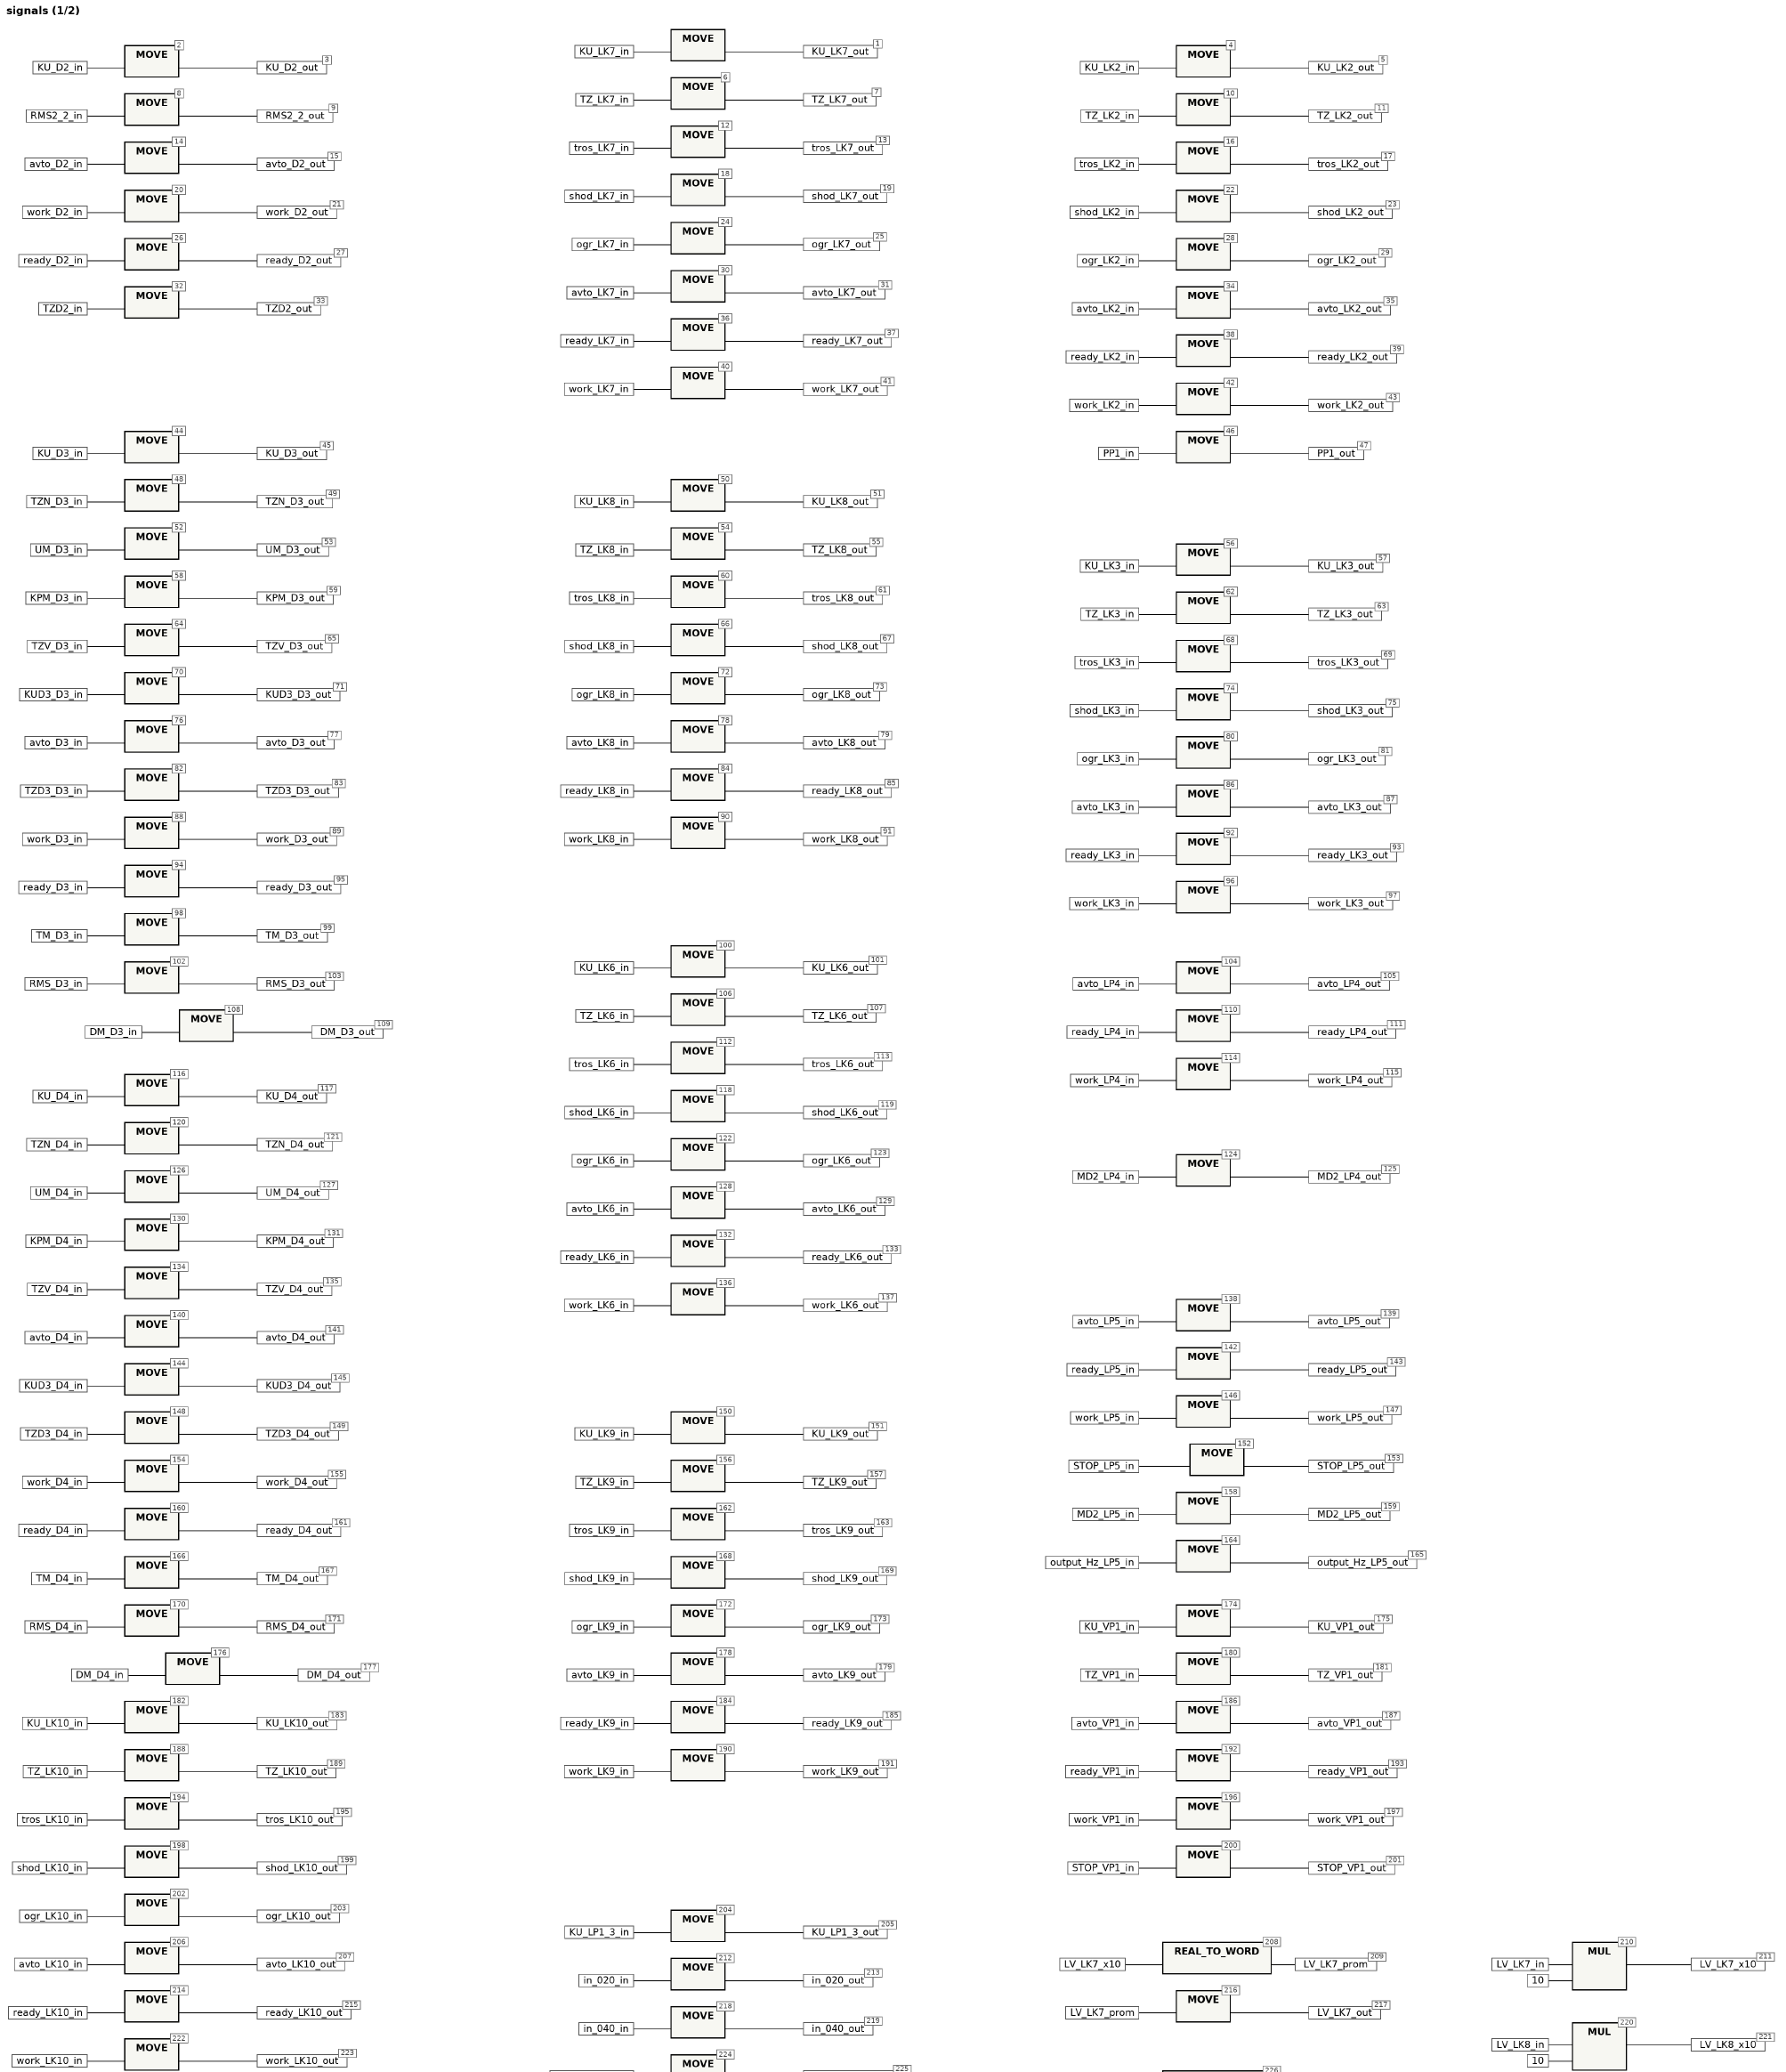
[picture p55: signals (CFC)]
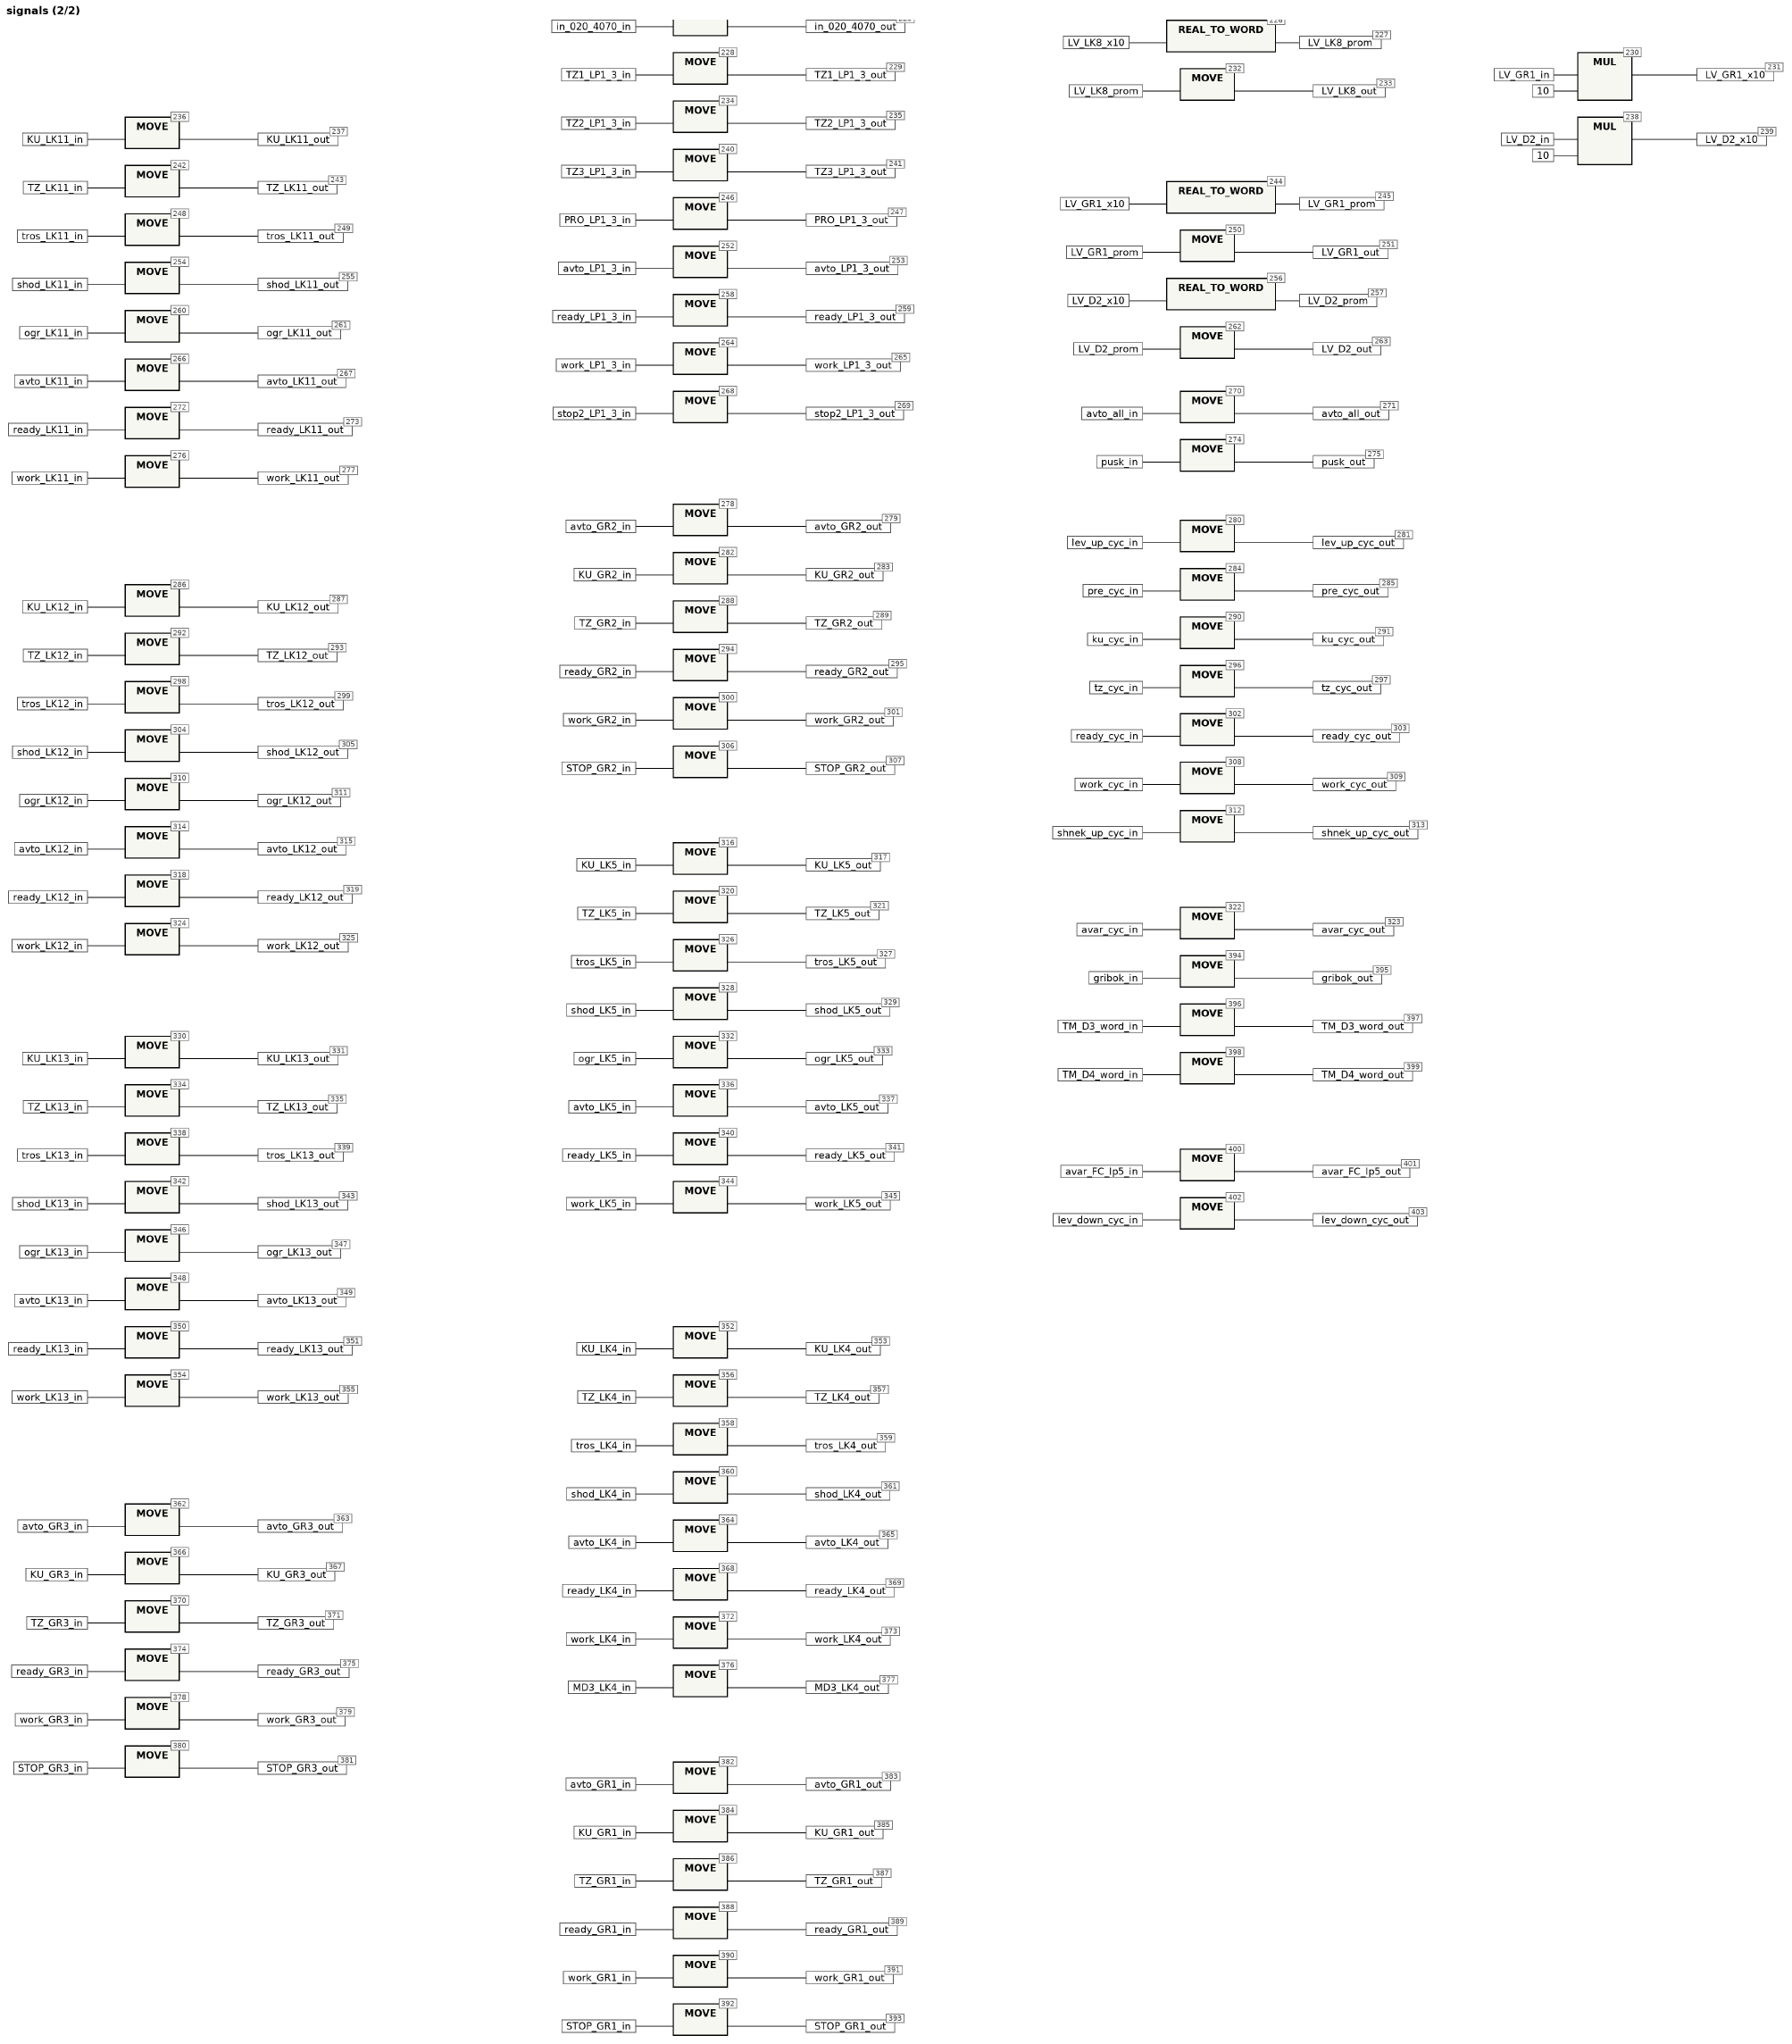
_CFC_ (* Continuous Function Chart, elements in execution order *)
#0 MOVE(KU_LK7_in)
#1 KU_LK7_out <= #0
#2 MOVE(KU_D2_in)
#3 KU_D2_out <= #2
#4 MOVE(KU_LK2_in)
#5 KU_LK2_out <= #4
#6 MOVE(TZ_LK7_in)
#7 TZ_LK7_out <= #6
#8 MOVE(RMS2_2_in)
#9 RMS2_2_out <= #8
#10 MOVE(TZ_LK2_in)
#11 TZ_LK2_out <= #10
#12 MOVE(tros_LK7_in)
#13 tros_LK7_out <= #12
#14 MOVE(avto_D2_in)
#15 avto_D2_out <= #14
#16 MOVE(tros_LK2_in)
#17 tros_LK2_out <= #16
#18 MOVE(shod_LK7_in)
#19 shod_LK7_out <= #18
#20 MOVE(work_D2_in)
#21 work_D2_out <= #20
#22 MOVE(shod_LK2_in)
#23 shod_LK2_out <= #22
#24 MOVE(ogr_LK7_in)
#25 ogr_LK7_out <= #24
#26 MOVE(ready_D2_in)
#27 ready_D2_out <= #26
#28 MOVE(ogr_LK2_in)
#29 ogr_LK2_out <= #28
#30 MOVE(avto_LK7_in)
#31 avto_LK7_out <= #30
#32 MOVE(TZD2_in)
#33 TZD2_out <= #32
#34 MOVE(avto_LK2_in)
#35 avto_LK2_out <= #34
#36 MOVE(ready_LK7_in)
#37 ready_LK7_out <= #36
#38 MOVE(ready_LK2_in)
#39 ready_LK2_out <= #38
#40 MOVE(work_LK7_in)
#41 work_LK7_out <= #40
#42 MOVE(work_LK2_in)
#43 work_LK2_out <= #42
#44 MOVE(KU_D3_in)
#45 KU_D3_out <= #44
#46 MOVE(PP1_in)
#47 PP1_out <= #46
#48 MOVE(TZN_D3_in)
#49 TZN_D3_out <= #48
#50 MOVE(KU_LK8_in)
#51 KU_LK8_out <= #50
#52 MOVE(UM_D3_in)
#53 UM_D3_out <= #52
#54 MOVE(TZ_LK8_in)
#55 TZ_LK8_out <= #54
#56 MOVE(KU_LK3_in)
#57 KU_LK3_out <= #56
#58 MOVE(KPM_D3_in)
#59 KPM_D3_out <= #58
#60 MOVE(tros_LK8_in)
#61 tros_LK8_out <= #60
#62 MOVE(TZ_LK3_in)
#63 TZ_LK3_out <= #62
#64 MOVE(TZV_D3_in)
#65 TZV_D3_out <= #64
#66 MOVE(shod_LK8_in)
#67 shod_LK8_out <= #66
#68 MOVE(tros_LK3_in)
#69 tros_LK3_out <= #68
#70 MOVE(KUD3_D3_in)
#71 KUD3_D3_out <= #70
#72 MOVE(ogr_LK8_in)
#73 ogr_LK8_out <= #72
#74 MOVE(shod_LK3_in)
#75 shod_LK3_out <= #74
#76 MOVE(avto_D3_in)
#77 avto_D3_out <= #76
#78 MOVE(avto_LK8_in)
#79 avto_LK8_out <= #78
#80 MOVE(ogr_LK3_in)
#81 ogr_LK3_out <= #80
#82 MOVE(TZD3_D3_in)
#83 TZD3_D3_out <= #82
#84 MOVE(ready_LK8_in)
#85 ready_LK8_out <= #84
#86 MOVE(avto_LK3_in)
#87 avto_LK3_out <= #86
#88 MOVE(work_D3_in)
#89 work_D3_out <= #88
#90 MOVE(work_LK8_in)
#91 work_LK8_out <= #90
#92 MOVE(ready_LK3_in)
#93 ready_LK3_out <= #92
#94 MOVE(ready_D3_in)
#95 ready_D3_out <= #94
#96 MOVE(work_LK3_in)
#97 work_LK3_out <= #96
#98 MOVE(TM_D3_in)
#99 TM_D3_out <= #98
#100 MOVE(KU_LK6_in)
#101 KU_LK6_out <= #100
#102 MOVE(RMS_D3_in)
#103 RMS_D3_out <= #102
#104 MOVE(avto_LP4_in)
#105 avto_LP4_out <= #104
#106 MOVE(TZ_LK6_in)
#107 TZ_LK6_out <= #106
#108 MOVE(DM_D3_in)
#109 DM_D3_out <= #108
#110 MOVE(ready_LP4_in)
#111 ready_LP4_out <= #110
#112 MOVE(tros_LK6_in)
#113 tros_LK6_out <= #112
#114 MOVE(work_LP4_in)
#115 work_LP4_out <= #114
#116 MOVE(KU_D4_in)
#117 KU_D4_out <= #116
#118 MOVE(shod_LK6_in)
#119 shod_LK6_out <= #118
#120 MOVE(TZN_D4_in)
#121 TZN_D4_out <= #120
#122 MOVE(ogr_LK6_in)
#123 ogr_LK6_out <= #122
#124 MOVE(MD2_LP4_in)
#125 MD2_LP4_out <= #124
#126 MOVE(UM_D4_in)
#127 UM_D4_out <= #126
#128 MOVE(avto_LK6_in)
#129 avto_LK6_out <= #128
#130 MOVE(KPM_D4_in)
#131 KPM_D4_out <= #130
#132 MOVE(ready_LK6_in)
#133 ready_LK6_out <= #132
#134 MOVE(TZV_D4_in)
#135 TZV_D4_out <= #134
#136 MOVE(work_LK6_in)
#137 work_LK6_out <= #136
#138 MOVE(avto_LP5_in)
#139 avto_LP5_out <= #138
#140 MOVE(avto_D4_in)
#141 avto_D4_out <= #140
#142 MOVE(ready_LP5_in)
#143 ready_LP5_out <= #142
#144 MOVE(KUD3_D4_in)
#145 KUD3_D4_out <= #144
#146 MOVE(work_LP5_in)
#147 work_LP5_out <= #146
#148 MOVE(TZD3_D4_in)
#149 TZD3_D4_out <= #148
#150 MOVE(KU_LK9_in)
#151 KU_LK9_out <= #150
#152 MOVE(STOP_LP5_in)
#153 STOP_LP5_out <= #152
#154 MOVE(work_D4_in)
#155 work_D4_out <= #154
#156 MOVE(TZ_LK9_in)
#157 TZ_LK9_out <= #156
#158 MOVE(MD2_LP5_in)
#159 MD2_LP5_out <= #158
#160 MOVE(ready_D4_in)
#161 ready_D4_out <= #160
#162 MOVE(tros_LK9_in)
#163 tros_LK9_out <= #162
#164 MOVE(output_Hz_LP5_in)
#165 output_Hz_LP5_out <= #164
#166 MOVE(TM_D4_in)
#167 TM_D4_out <= #166
#168 MOVE(shod_LK9_in)
#169 shod_LK9_out <= #168
#170 MOVE(RMS_D4_in)
#171 RMS_D4_out <= #170
#172 MOVE(ogr_LK9_in)
#173 ogr_LK9_out <= #172
#174 MOVE(KU_VP1_in)
#175 KU_VP1_out <= #174
#176 MOVE(DM_D4_in)
#177 DM_D4_out <= #176
#178 MOVE(avto_LK9_in)
#179 avto_LK9_out <= #178
#180 MOVE(TZ_VP1_in)
#181 TZ_VP1_out <= #180
#182 MOVE(KU_LK10_in)
#183 KU_LK10_out <= #182
#184 MOVE(ready_LK9_in)
#185 ready_LK9_out <= #184
#186 MOVE(avto_VP1_in)
#187 avto_VP1_out <= #186
#188 MOVE(TZ_LK10_in)
#189 TZ_LK10_out <= #188
#190 MOVE(work_LK9_in)
#191 work_LK9_out <= #190
#192 MOVE(ready_VP1_in)
#193 ready_VP1_out <= #192
#194 MOVE(tros_LK10_in)
#195 tros_LK10_out <= #194
#196 MOVE(work_VP1_in)
#197 work_VP1_out <= #196
#198 MOVE(shod_LK10_in)
#199 shod_LK10_out <= #198
#200 MOVE(STOP_VP1_in)
#201 STOP_VP1_out <= #200
#202 MOVE(ogr_LK10_in)
#203 ogr_LK10_out <= #202
#204 MOVE(KU_LP1_3_in)
#205 KU_LP1_3_out <= #204
#206 MOVE(avto_LK10_in)
#207 avto_LK10_out <= #206
#208 REAL_TO_WORD(LV_LK7_x10)
#209 LV_LK7_prom <= #208
#210 MUL(LV_LK7_in, 10)
#211 LV_LK7_x10 <= #210
#212 MOVE(in_020_in)
#213 in_020_out <= #212
#214 MOVE(ready_LK10_in)
#215 ready_LK10_out <= #214
#216 MOVE(LV_LK7_prom)
#217 LV_LK7_out <= #216
#218 MOVE(in_040_in)
#219 in_040_out <= #218
#220 MUL(LV_LK8_in, 10)
#221 LV_LK8_x10 <= #220
#222 MOVE(work_LK10_in)
#223 work_LK10_out <= #222
#224 MOVE(in_020_4070_in)
#225 in_020_4070_out <= #224
#226 REAL_TO_WORD(LV_LK8_x10)
#227 LV_LK8_prom <= #226
#228 MOVE(TZ1_LP1_3_in)
#229 TZ1_LP1_3_out <= #228
#230 MUL(LV_GR1_in, 10)
#231 LV_GR1_x10 <= #230
#232 MOVE(LV_LK8_prom)
#233 LV_LK8_out <= #232
#234 MOVE(TZ2_LP1_3_in)
#235 TZ2_LP1_3_out <= #234
#236 MOVE(KU_LK11_in)
#237 KU_LK11_out <= #236
#238 MUL(LV_D2_in, 10)
#239 LV_D2_x10 <= #238
#240 MOVE(TZ3_LP1_3_in)
#241 TZ3_LP1_3_out <= #240
#242 MOVE(TZ_LK11_in)
#243 TZ_LK11_out <= #242
#244 REAL_TO_WORD(LV_GR1_x10)
#245 LV_GR1_prom <= #244
#246 MOVE(PRO_LP1_3_in)
#247 PRO_LP1_3_out <= #246
#248 MOVE(tros_LK11_in)
#249 tros_LK11_out <= #248
#250 MOVE(LV_GR1_prom)
#251 LV_GR1_out <= #250
#252 MOVE(avto_LP1_3_in)
#253 avto_LP1_3_out <= #252
#254 MOVE(shod_LK11_in)
#255 shod_LK11_out <= #254
#256 REAL_TO_WORD(LV_D2_x10)
#257 LV_D2_prom <= #256
#258 MOVE(ready_LP1_3_in)
#259 ready_LP1_3_out <= #258
#260 MOVE(ogr_LK11_in)
#261 ogr_LK11_out <= #260
#262 MOVE(LV_D2_prom)
#263 LV_D2_out <= #262
#264 MOVE(work_LP1_3_in)
#265 work_LP1_3_out <= #264
#266 MOVE(avto_LK11_in)
#267 avto_LK11_out <= #266
#268 MOVE(stop2_LP1_3_in)
#269 stop2_LP1_3_out <= #268
#270 MOVE(avto_all_in)
#271 avto_all_out <= #270
#272 MOVE(ready_LK11_in)
#273 ready_LK11_out <= #272
#274 MOVE(pusk_in)
#275 pusk_out <= #274
#276 MOVE(work_LK11_in)
#277 work_LK11_out <= #276
#278 MOVE(avto_GR2_in)
#279 avto_GR2_out <= #278
#280 MOVE(lev_up_cyc_in)
#281 lev_up_cyc_out <= #280
#282 MOVE(KU_GR2_in)
#283 KU_GR2_out <= #282
#284 MOVE(pre_cyc_in)
#285 pre_cyc_out <= #284
#286 MOVE(KU_LK12_in)
#287 KU_LK12_out <= #286
#288 MOVE(TZ_GR2_in)
#289 TZ_GR2_out <= #288
#290 MOVE(ku_cyc_in)
#291 ku_cyc_out <= #290
#292 MOVE(TZ_LK12_in)
#293 TZ_LK12_out <= #292
#294 MOVE(ready_GR2_in)
#295 ready_GR2_out <= #294
#296 MOVE(tz_cyc_in)
#297 tz_cyc_out <= #296
#298 MOVE(tros_LK12_in)
#299 tros_LK12_out <= #298
#300 MOVE(work_GR2_in)
#301 work_GR2_out <= #300
#302 MOVE(ready_cyc_in)
#303 ready_cyc_out <= #302
#304 MOVE(shod_LK12_in)
#305 shod_LK12_out <= #304
#306 MOVE(STOP_GR2_in)
#307 STOP_GR2_out <= #306
#308 MOVE(work_cyc_in)
#309 work_cyc_out <= #308
#310 MOVE(ogr_LK12_in)
#311 ogr_LK12_out <= #310
#312 MOVE(shnek_up_cyc_in)
#313 shnek_up_cyc_out <= #312
#314 MOVE(avto_LK12_in)
#315 avto_LK12_out <= #314
#316 MOVE(KU_LK5_in)
#317 KU_LK5_out <= #316
#318 MOVE(ready_LK12_in)
#319 ready_LK12_out <= #318
#320 MOVE(TZ_LK5_in)
#321 TZ_LK5_out <= #320
#322 MOVE(avar_cyc_in)
#323 avar_cyc_out <= #322
#324 MOVE(work_LK12_in)
#325 work_LK12_out <= #324
#326 MOVE(tros_LK5_in)
#327 tros_LK5_out <= #326
#328 MOVE(shod_LK5_in)
#329 shod_LK5_out <= #328
#330 MOVE(KU_LK13_in)
#331 KU_LK13_out <= #330
#332 MOVE(ogr_LK5_in)
#333 ogr_LK5_out <= #332
#334 MOVE(TZ_LK13_in)
#335 TZ_LK13_out <= #334
#336 MOVE(avto_LK5_in)
#337 avto_LK5_out <= #336
#338 MOVE(tros_LK13_in)
#339 tros_LK13_out <= #338
#340 MOVE(ready_LK5_in)
#341 ready_LK5_out <= #340
#342 MOVE(shod_LK13_in)
#343 shod_LK13_out <= #342
#344 MOVE(work_LK5_in)
#345 work_LK5_out <= #344
#346 MOVE(ogr_LK13_in)
#347 ogr_LK13_out <= #346
#348 MOVE(avto_LK13_in)
#349 avto_LK13_out <= #348
#350 MOVE(ready_LK13_in)
#351 ready_LK13_out <= #350
#352 MOVE(KU_LK4_in)
#353 KU_LK4_out <= #352
#354 MOVE(work_LK13_in)
#355 work_LK13_out <= #354
#356 MOVE(TZ_LK4_in)
#357 TZ_LK4_out <= #356
#358 MOVE(tros_LK4_in)
#359 tros_LK4_out <= #358
#360 MOVE(shod_LK4_in)
#361 shod_LK4_out <= #360
#362 MOVE(avto_GR3_in)
#363 avto_GR3_out <= #362
#364 MOVE(avto_LK4_in)
#365 avto_LK4_out <= #364
#366 MOVE(KU_GR3_in)
#367 KU_GR3_out <= #366
#368 MOVE(ready_LK4_in)
#369 ready_LK4_out <= #368
#370 MOVE(TZ_GR3_in)
#371 TZ_GR3_out <= #370
#372 MOVE(work_LK4_in)
#373 work_LK4_out <= #372
#374 MOVE(ready_GR3_in)
#375 ready_GR3_out <= #374
#376 MOVE(MD3_LK4_in)
#377 MD3_LK4_out <= #376
#378 MOVE(work_GR3_in)
#379 work_GR3_out <= #378
#380 MOVE(STOP_GR3_in)
#381 STOP_GR3_out <= #380
#382 MOVE(avto_GR1_in)
#383 avto_GR1_out <= #382
#384 MOVE(KU_GR1_in)
#385 KU_GR1_out <= #384
#386 MOVE(TZ_GR1_in)
#387 TZ_GR1_out <= #386
#388 MOVE(ready_GR1_in)
#389 ready_GR1_out <= #388
#390 MOVE(work_GR1_in)
#391 work_GR1_out <= #390
#392 MOVE(STOP_GR1_in)
#393 STOP_GR1_out <= #392
#394 MOVE(gribok_in)
#395 gribok_out <= #394
#396 MOVE(TM_D3_word_in)
#397 TM_D3_word_out <= #396
#398 MOVE(TM_D4_word_in)
#399 TM_D4_word_out <= #398
#400 MOVE(avar_FC_lp5_in)
#401 avar_FC_lp5_out <= #400
#402 MOVE(lev_down_cyc_in)
#403 lev_down_cyc_out <= #402
_END_CFC_
(* the same logic as Structured Text *)
KU_LK7_out := KU_LK7_in;
KU_D2_out := KU_D2_in;
KU_LK2_out := KU_LK2_in;
TZ_LK7_out := TZ_LK7_in;
RMS2_2_out := RMS2_2_in;
TZ_LK2_out := TZ_LK2_in;
tros_LK7_out := tros_LK7_in;
avto_D2_out := avto_D2_in;
tros_LK2_out := tros_LK2_in;
shod_LK7_out := shod_LK7_in;
work_D2_out := work_D2_in;
shod_LK2_out := shod_LK2_in;
ogr_LK7_out := ogr_LK7_in;
ready_D2_out := ready_D2_in;
ogr_LK2_out := ogr_LK2_in;
avto_LK7_out := avto_LK7_in;
TZD2_out := TZD2_in;
avto_LK2_out := avto_LK2_in;
ready_LK7_out := ready_LK7_in;
ready_LK2_out := ready_LK2_in;
work_LK7_out := work_LK7_in;
work_LK2_out := work_LK2_in;
KU_D3_out := KU_D3_in;
PP1_out := PP1_in;
TZN_D3_out := TZN_D3_in;
KU_LK8_out := KU_LK8_in;
UM_D3_out := UM_D3_in;
TZ_LK8_out := TZ_LK8_in;
KU_LK3_out := KU_LK3_in;
KPM_D3_out := KPM_D3_in;
tros_LK8_out := tros_LK8_in;
TZ_LK3_out := TZ_LK3_in;
TZV_D3_out := TZV_D3_in;
shod_LK8_out := shod_LK8_in;
tros_LK3_out := tros_LK3_in;
KUD3_D3_out := KUD3_D3_in;
ogr_LK8_out := ogr_LK8_in;
shod_LK3_out := shod_LK3_in;
avto_D3_out := avto_D3_in;
avto_LK8_out := avto_LK8_in;
ogr_LK3_out := ogr_LK3_in;
TZD3_D3_out := TZD3_D3_in;
ready_LK8_out := ready_LK8_in;
avto_LK3_out := avto_LK3_in;
work_D3_out := work_D3_in;
work_LK8_out := work_LK8_in;
ready_LK3_out := ready_LK3_in;
ready_D3_out := ready_D3_in;
work_LK3_out := work_LK3_in;
TM_D3_out := TM_D3_in;
KU_LK6_out := KU_LK6_in;
RMS_D3_out := RMS_D3_in;
avto_LP4_out := avto_LP4_in;
TZ_LK6_out := TZ_LK6_in;
DM_D3_out := DM_D3_in;
ready_LP4_out := ready_LP4_in;
tros_LK6_out := tros_LK6_in;
work_LP4_out := work_LP4_in;
KU_D4_out := KU_D4_in;
shod_LK6_out := shod_LK6_in;
TZN_D4_out := TZN_D4_in;
ogr_LK6_out := ogr_LK6_in;
MD2_LP4_out := MD2_LP4_in;
UM_D4_out := UM_D4_in;
avto_LK6_out := avto_LK6_in;
KPM_D4_out := KPM_D4_in;
ready_LK6_out := ready_LK6_in;
TZV_D4_out := TZV_D4_in;
work_LK6_out := work_LK6_in;
avto_LP5_out := avto_LP5_in;
avto_D4_out := avto_D4_in;
ready_LP5_out := ready_LP5_in;
KUD3_D4_out := KUD3_D4_in;
work_LP5_out := work_LP5_in;
TZD3_D4_out := TZD3_D4_in;
KU_LK9_out := KU_LK9_in;
STOP_LP5_out := STOP_LP5_in;
work_D4_out := work_D4_in;
TZ_LK9_out := TZ_LK9_in;
MD2_LP5_out := MD2_LP5_in;
ready_D4_out := ready_D4_in;
tros_LK9_out := tros_LK9_in;
output_Hz_LP5_out := output_Hz_LP5_in;
TM_D4_out := TM_D4_in;
shod_LK9_out := shod_LK9_in;
RMS_D4_out := RMS_D4_in;
ogr_LK9_out := ogr_LK9_in;
KU_VP1_out := KU_VP1_in;
DM_D4_out := DM_D4_in;
avto_LK9_out := avto_LK9_in;
TZ_VP1_out := TZ_VP1_in;
KU_LK10_out := KU_LK10_in;
ready_LK9_out := ready_LK9_in;
avto_VP1_out := avto_VP1_in;
TZ_LK10_out := TZ_LK10_in;
work_LK9_out := work_LK9_in;
ready_VP1_out := ready_VP1_in;
tros_LK10_out := tros_LK10_in;
work_VP1_out := work_VP1_in;
shod_LK10_out := shod_LK10_in;
STOP_VP1_out := STOP_VP1_in;
ogr_LK10_out := ogr_LK10_in;
KU_LP1_3_out := KU_LP1_3_in;
avto_LK10_out := avto_LK10_in;
LV_LK7_prom := REAL_TO_WORD(LV_LK7_x10);
LV_LK7_x10 := LV_LK7_in * 10;
in_020_out := in_020_in;
ready_LK10_out := ready_LK10_in;
LV_LK7_out := LV_LK7_prom;
in_040_out := in_040_in;
LV_LK8_x10 := LV_LK8_in * 10;
work_LK10_out := work_LK10_in;
in_020_4070_out := in_020_4070_in;
LV_LK8_prom := REAL_TO_WORD(LV_LK8_x10);
TZ1_LP1_3_out := TZ1_LP1_3_in;
LV_GR1_x10 := LV_GR1_in * 10;
LV_LK8_out := LV_LK8_prom;
TZ2_LP1_3_out := TZ2_LP1_3_in;
KU_LK11_out := KU_LK11_in;
LV_D2_x10 := LV_D2_in * 10;
TZ3_LP1_3_out := TZ3_LP1_3_in;
TZ_LK11_out := TZ_LK11_in;
LV_GR1_prom := REAL_TO_WORD(LV_GR1_x10);
PRO_LP1_3_out := PRO_LP1_3_in;
tros_LK11_out := tros_LK11_in;
LV_GR1_out := LV_GR1_prom;
avto_LP1_3_out := avto_LP1_3_in;
shod_LK11_out := shod_LK11_in;
LV_D2_prom := REAL_TO_WORD(LV_D2_x10);
ready_LP1_3_out := ready_LP1_3_in;
ogr_LK11_out := ogr_LK11_in;
LV_D2_out := LV_D2_prom;
work_LP1_3_out := work_LP1_3_in;
avto_LK11_out := avto_LK11_in;
stop2_LP1_3_out := stop2_LP1_3_in;
avto_all_out := avto_all_in;
ready_LK11_out := ready_LK11_in;
pusk_out := pusk_in;
work_LK11_out := work_LK11_in;
avto_GR2_out := avto_GR2_in;
lev_up_cyc_out := lev_up_cyc_in;
KU_GR2_out := KU_GR2_in;
pre_cyc_out := pre_cyc_in;
KU_LK12_out := KU_LK12_in;
TZ_GR2_out := TZ_GR2_in;
ku_cyc_out := ku_cyc_in;
TZ_LK12_out := TZ_LK12_in;
ready_GR2_out := ready_GR2_in;
tz_cyc_out := tz_cyc_in;
tros_LK12_out := tros_LK12_in;
work_GR2_out := work_GR2_in;
ready_cyc_out := ready_cyc_in;
shod_LK12_out := shod_LK12_in;
STOP_GR2_out := STOP_GR2_in;
work_cyc_out := work_cyc_in;
ogr_LK12_out := ogr_LK12_in;
shnek_up_cyc_out := shnek_up_cyc_in;
avto_LK12_out := avto_LK12_in;
KU_LK5_out := KU_LK5_in;
ready_LK12_out := ready_LK12_in;
TZ_LK5_out := TZ_LK5_in;
avar_cyc_out := avar_cyc_in;
work_LK12_out := work_LK12_in;
tros_LK5_out := tros_LK5_in;
shod_LK5_out := shod_LK5_in;
KU_LK13_out := KU_LK13_in;
ogr_LK5_out := ogr_LK5_in;
TZ_LK13_out := TZ_LK13_in;
avto_LK5_out := avto_LK5_in;
tros_LK13_out := tros_LK13_in;
ready_LK5_out := ready_LK5_in;
shod_LK13_out := shod_LK13_in;
work_LK5_out := work_LK5_in;
ogr_LK13_out := ogr_LK13_in;
avto_LK13_out := avto_LK13_in;
ready_LK13_out := ready_LK13_in;
KU_LK4_out := KU_LK4_in;
work_LK13_out := work_LK13_in;
TZ_LK4_out := TZ_LK4_in;
tros_LK4_out := tros_LK4_in;
shod_LK4_out := shod_LK4_in;
avto_GR3_out := avto_GR3_in;
avto_LK4_out := avto_LK4_in;
KU_GR3_out := KU_GR3_in;
ready_LK4_out := ready_LK4_in;
TZ_GR3_out := TZ_GR3_in;
work_LK4_out := work_LK4_in;
ready_GR3_out := ready_GR3_in;
MD3_LK4_out := MD3_LK4_in;
work_GR3_out := work_GR3_in;
STOP_GR3_out := STOP_GR3_in;
avto_GR1_out := avto_GR1_in;
KU_GR1_out := KU_GR1_in;
TZ_GR1_out := TZ_GR1_in;
ready_GR1_out := ready_GR1_in;
work_GR1_out := work_GR1_in;
STOP_GR1_out := STOP_GR1_in;
gribok_out := gribok_in;
TM_D3_word_out := TM_D3_word_in;
TM_D4_word_out := TM_D4_word_in;
avar_FC_lp5_out := avar_FC_lp5_in;
lev_down_cyc_out := lev_down_cyc_in;
END_FUNCTION_BLOCK

(* POU alarm, CFC *)
FUNCTION_BLOCK alarm (*функциональный блок, который проверяет наличие управляющего модуля в сети*)
VAR_INPUT
	adress_in_rs2: DWORD; (*входящий адрес опращиваемого устройства в RS485-2*)
	error_81_in_rs2: WORD; (*отслеживание наличия ошибки связи в RS485-2*)
	adress_in_rs1: DWORD; (*входящий адрес опращиваемого устройства в RS485-1*)
	error_81_in_rs1: WORD; (*отслеживание наличия ошибки связи в RS485-1*)
END_VAR
VAR_OUTPUT
	err_LK10: BOOL;
	err_LK11: BOOL;
	err_LK12: BOOL;
	err_LK13: BOOL;
	err_GR3: BOOL;
	err_LK7: BOOL;
	err_LK8: BOOL;
	err_LK6: BOOL;
	err_LK9: BOOL;
	err_LP1_3_mod1: BOOL;
	err_LP1_3_mod2: BOOL;
	err_GR2: BOOL;
	err_LK5: BOOL;
	err_LP4: BOOL;
	err_LP5: BOOL;
	err_LK4: BOOL;
	err_GR1: BOOL;
	err_LK2: BOOL;
	err_LK3: BOOL;
	err_VP1: BOOL;
	err_D3_mod1: BOOL;
	err_D3_mod2: BOOL;
	err_D4_mod1: BOOL;
	err_D4_mod2: BOOL;
	err_D2: BOOL;
	err_cyc1: BOOL;
	err_cyc2: BOOL;
	err_lp4_temp: BOOL;
	err_d3_temp: BOOL;
	err_d4_temp: BOOL;
	err_vp1_temp: BOOL;
END_VAR
VAR
	err_true_rs1: BOOL;
	err_false_rs1: BOOL;
	err_true_rs2: BOOL;
	err_false_rs2: BOOL;
	trig_LK10: RS;
	ton_lk10: TON;
	trig_LK11: RS;
	ton_lk11: TON;
	trig_LK12: RS;
	ton_lk12: TON;
	trig_LK13: RS;
	ton_lk13: TON;
	trig_gr3: RS;
	ton_gr3: TON;
	trig_lk7: RS;
	ton_lk7: TON;
	trig_lk8: RS;
	ton_lk8: TON;
	trig_lk6: RS;
	ton_lk6: TON;
	trig_LK9: RS;
	ton_lk9: TON;
	trig_LP1_3_1: RS;
	ton_LP1_3_1: TON;
	trig_LP1_3_2: RS;
	ton_LP1_3_2: TON;
	trig_GR2: RS;
	ton_GR2: TON;
	trig_lk5: RS;
	ton_lk5: TON;
	trig_lp4: RS;
	ton_lp4: TON;
	trig_lp5: RS;
	ton_lp5: TON;
	trig_lk4: RS;
	ton_lk4: TON;
	trig_gr1: RS;
	ton_gr1: TON;
	trig_lk2: RS;
	ton_lk2: TON;
	trig_lk3: RS;
	ton_lk3: TON;
	trig_vp1: RS;
	ton_vp1: TON;
	trig_d3_1: RS;
	ton_d3_1: TON;
	trig_d3_2: RS;
	ton_d3_2: TON;
	trig_d4_1: RS;
	ton_d4_1: TON;
	trig_d4_2: RS;
	ton_d4_2: TON;
	trig_d2: RS;
	ton_d2: TON;
	t: TIME:= t#2s;
	trig_cyc: RS;
	ton_cyc: TON;
	trig_cyc1: RS;
	ton_cyc1: TON;
	trig_lp4_temp: RS;
	ton_lp4_temp: TON;
	trig_d3_temp: RS;
	ton_d3_temp: TON;
	trig_d4_temp: RS;
	ton_d4_temp: TON;
	trig_vp1_temp: RS;
	ton_vp1_temp: TON;
END_VAR
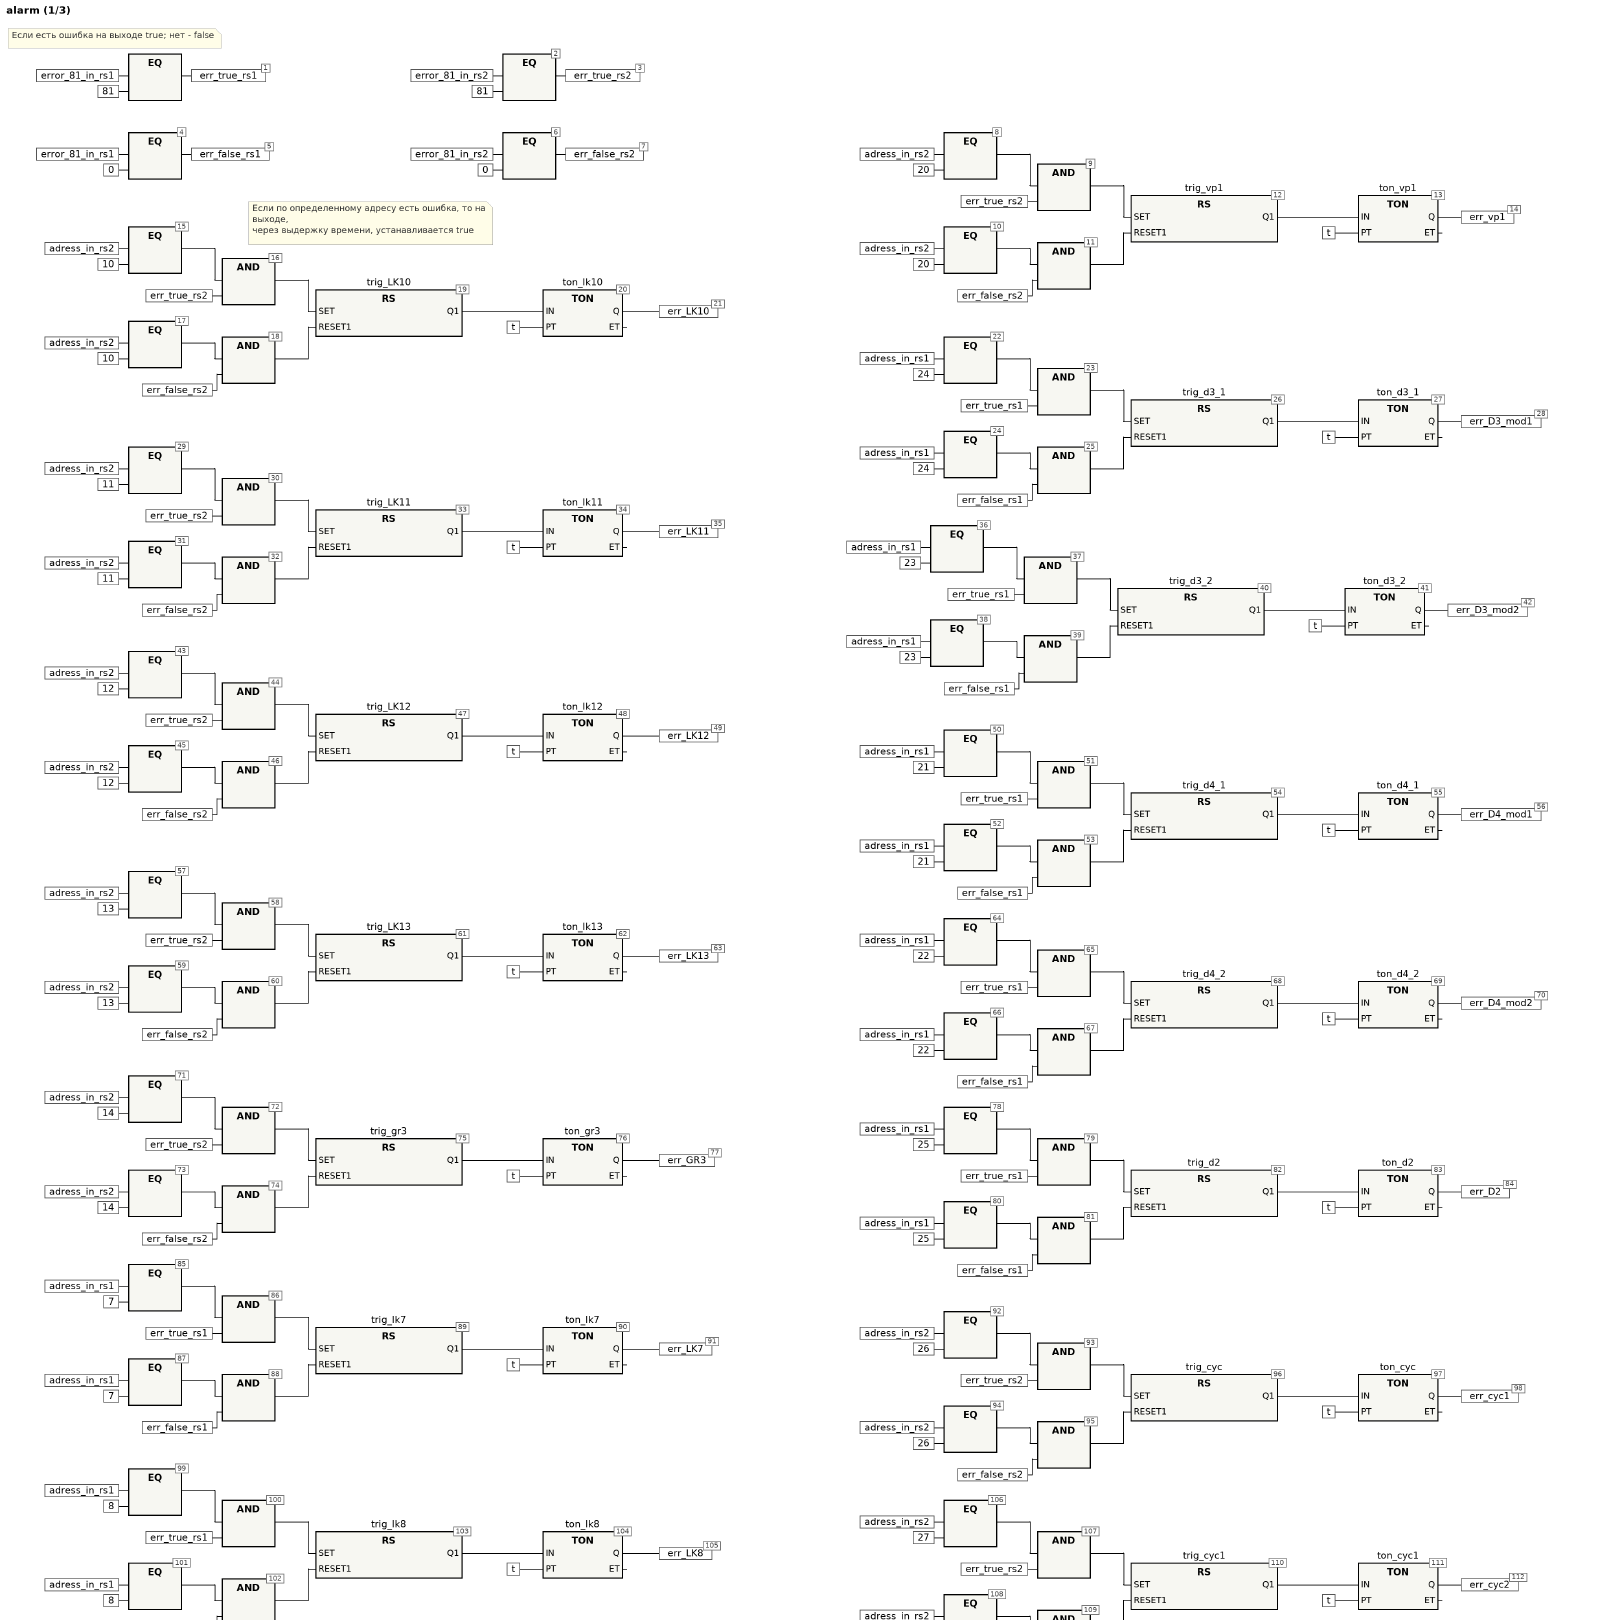
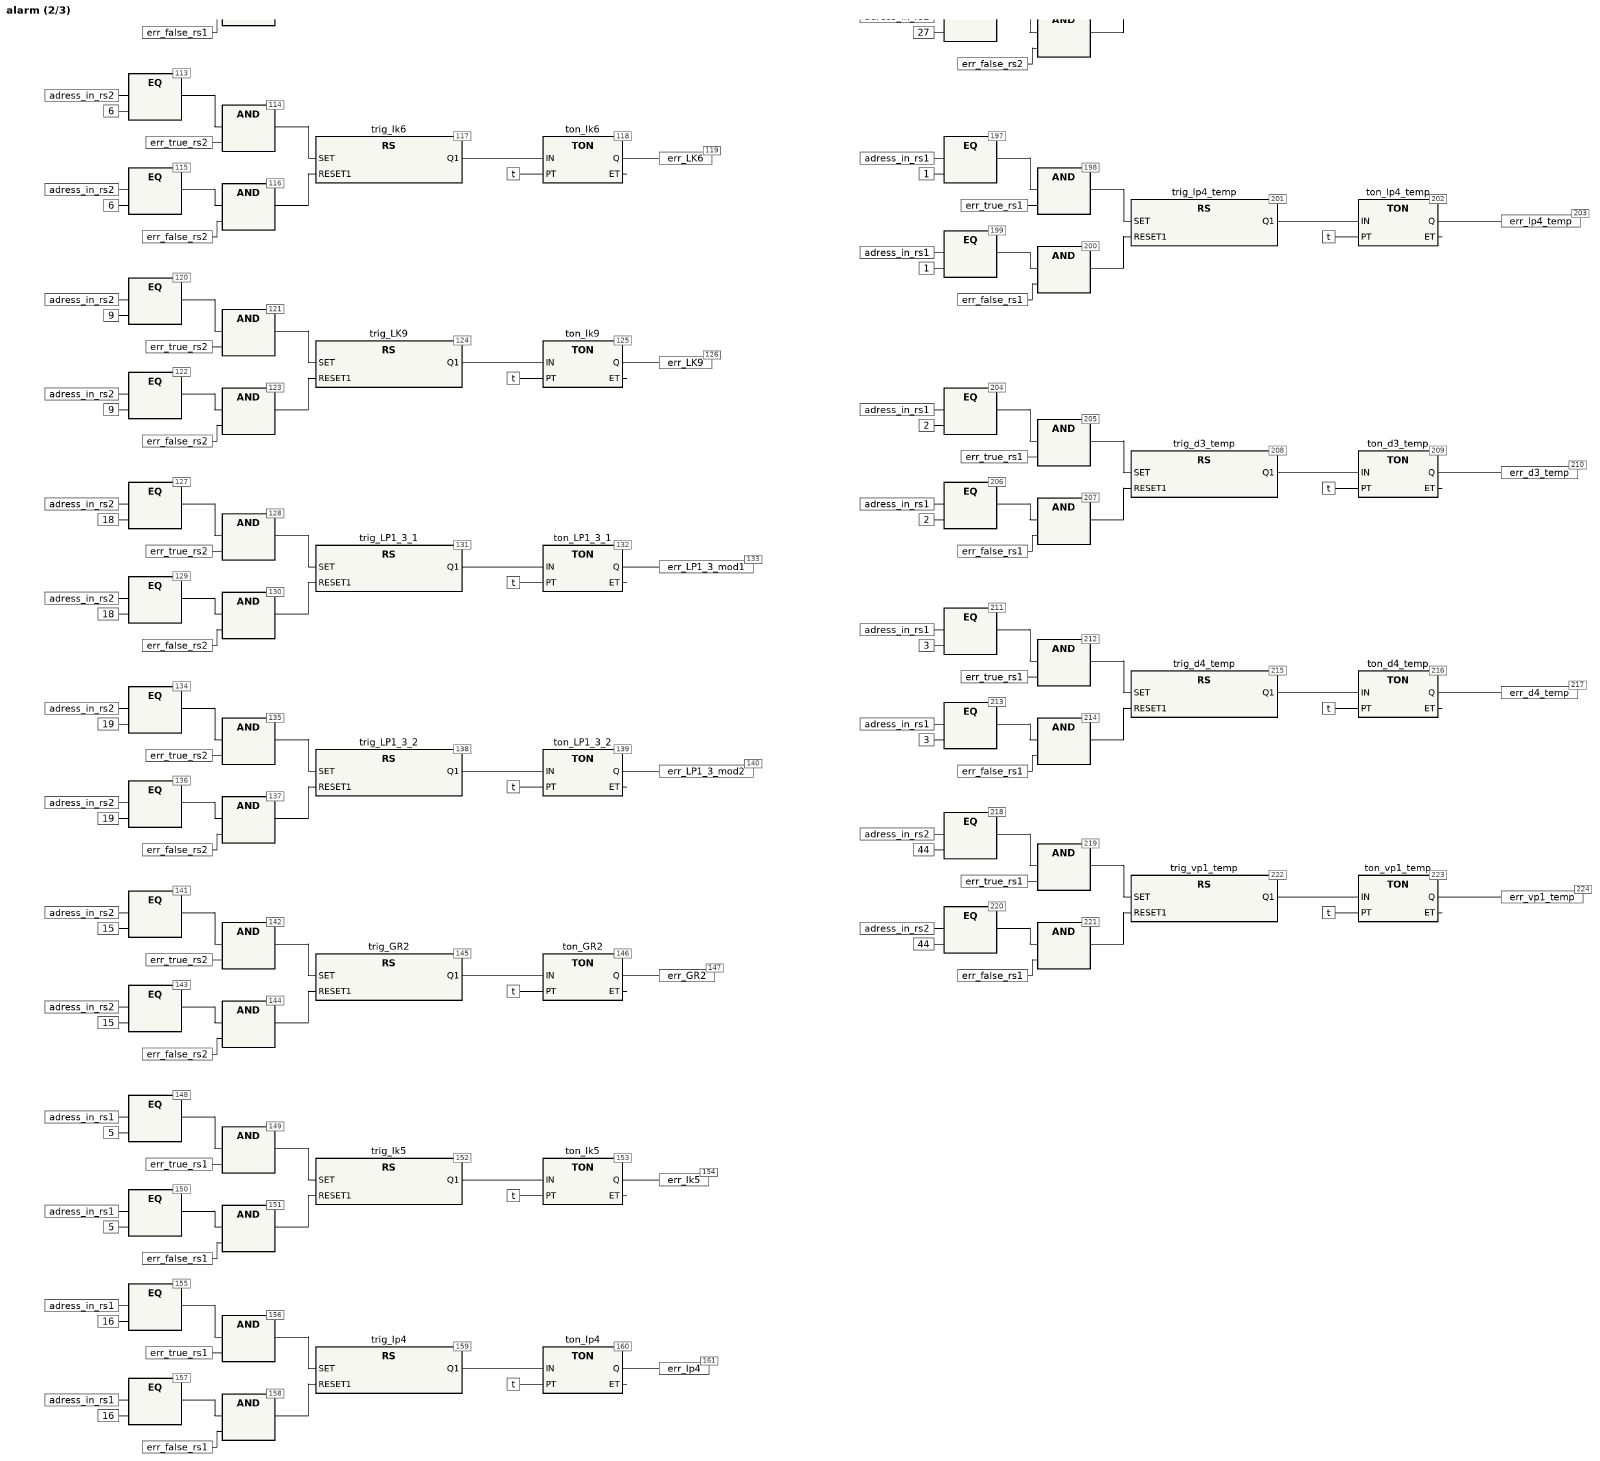
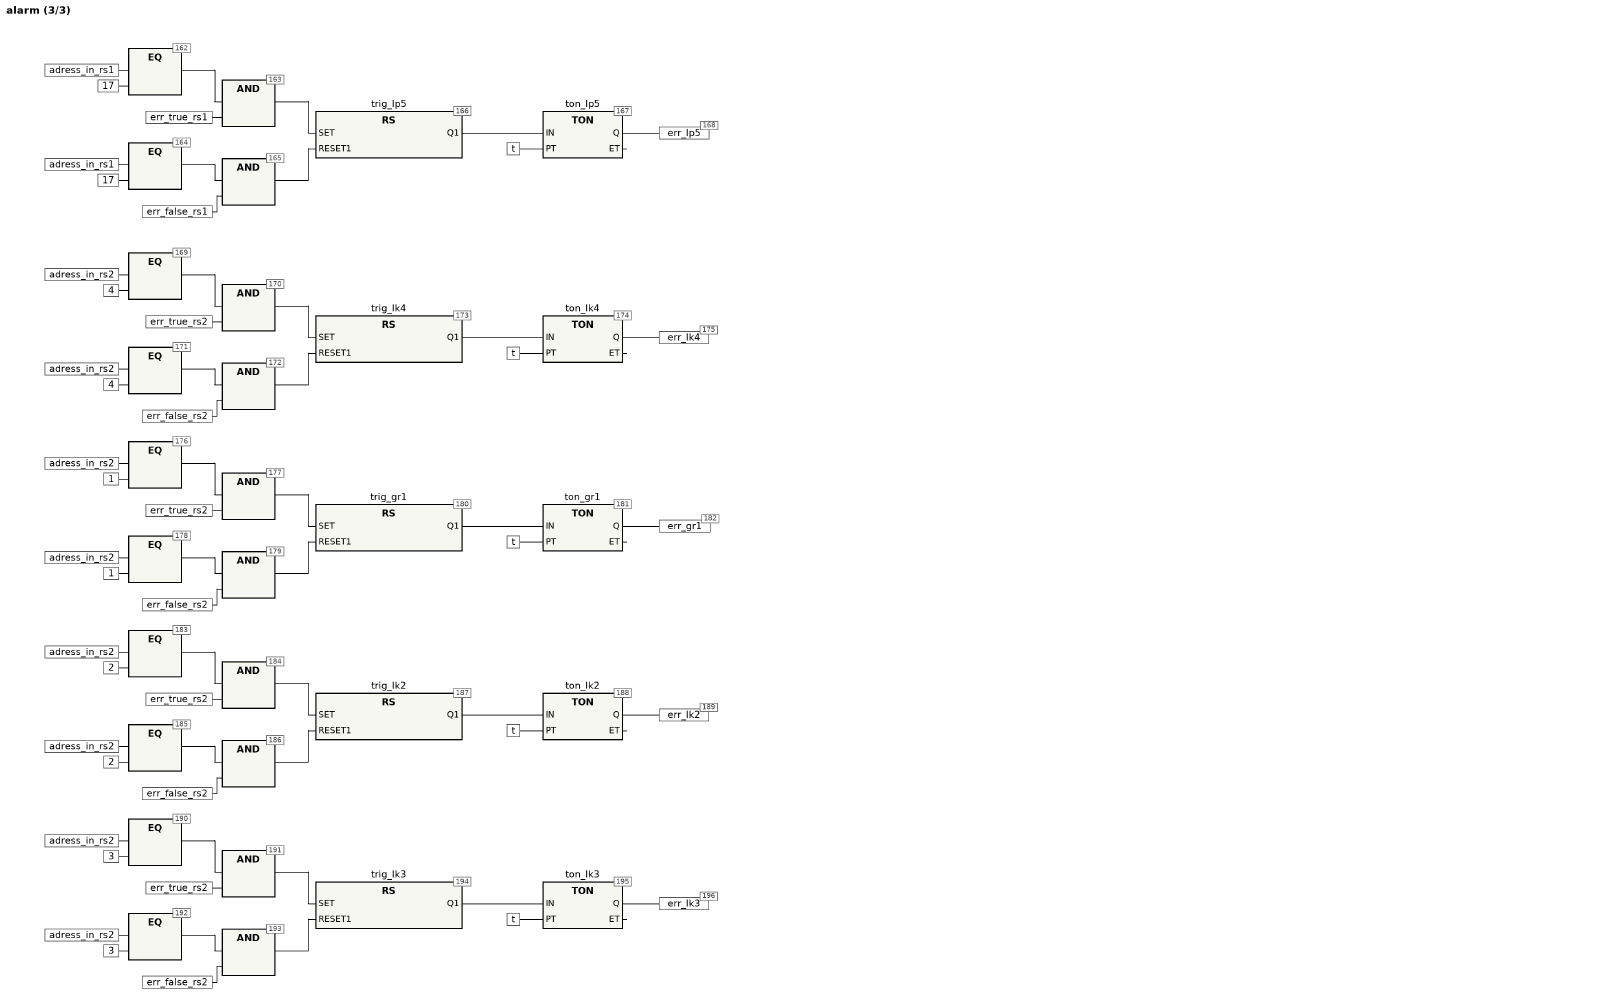
_CFC_ (* Continuous Function Chart, elements in execution order *)
(* Если есть ошибка на выходе true; нет - false *)
(* Если по определенному адресу есть ошибка, то на выходе, / через выдержку времени, устанавливается true *)
#0 EQ(error_81_in_rs1, 81)
#1 err_true_rs1 <= #0
#2 EQ(error_81_in_rs2, 81)
#3 err_true_rs2 <= #2
#4 EQ(error_81_in_rs1, 0)
#5 err_false_rs1 <= #4
#6 EQ(error_81_in_rs2, 0)
#7 err_false_rs2 <= #6
#8 EQ(adress_in_rs2, 20)
#9 AND(#8, err_true_rs2)
#10 EQ(adress_in_rs2, 20)
#11 AND(#10, err_false_rs2)
#12 trig_vp1:RS(SET: #9, RESET1: #11)
#13 ton_vp1:TON(IN: #12.Q1, PT: t)
#14 err_vp1 <= #13.Q
#15 EQ(adress_in_rs2, 10)
#16 AND(#15, err_true_rs2)
#17 EQ(adress_in_rs2, 10)
#18 AND(#17, err_false_rs2)
#19 trig_LK10:RS(SET: #16, RESET1: #18)
#20 ton_lk10:TON(IN: #19.Q1, PT: t)
#21 err_LK10 <= #20.Q
#22 EQ(adress_in_rs1, 24)
#23 AND(#22, err_true_rs1)
#24 EQ(adress_in_rs1, 24)
#25 AND(#24, err_false_rs1)
#26 trig_d3_1:RS(SET: #23, RESET1: #25)
#27 ton_d3_1:TON(IN: #26.Q1, PT: t)
#28 err_D3_mod1 <= #27.Q
#29 EQ(adress_in_rs2, 11)
#30 AND(#29, err_true_rs2)
#31 EQ(adress_in_rs2, 11)
#32 AND(#31, err_false_rs2)
#33 trig_LK11:RS(SET: #30, RESET1: #32)
#34 ton_lk11:TON(IN: #33.Q1, PT: t)
#35 err_LK11 <= #34.Q
#36 EQ(adress_in_rs1, 23)
#37 AND(#36, err_true_rs1)
#38 EQ(adress_in_rs1, 23)
#39 AND(#38, err_false_rs1)
#40 trig_d3_2:RS(SET: #37, RESET1: #39)
#41 ton_d3_2:TON(IN: #40.Q1, PT: t)
#42 err_D3_mod2 <= #41.Q
#43 EQ(adress_in_rs2, 12)
#44 AND(#43, err_true_rs2)
#45 EQ(adress_in_rs2, 12)
#46 AND(#45, err_false_rs2)
#47 trig_LK12:RS(SET: #44, RESET1: #46)
#48 ton_lk12:TON(IN: #47.Q1, PT: t)
#49 err_LK12 <= #48.Q
#50 EQ(adress_in_rs1, 21)
#51 AND(#50, err_true_rs1)
#52 EQ(adress_in_rs1, 21)
#53 AND(#52, err_false_rs1)
#54 trig_d4_1:RS(SET: #51, RESET1: #53)
#55 ton_d4_1:TON(IN: #54.Q1, PT: t)
#56 err_D4_mod1 <= #55.Q
#57 EQ(adress_in_rs2, 13)
#58 AND(#57, err_true_rs2)
#59 EQ(adress_in_rs2, 13)
#60 AND(#59, err_false_rs2)
#61 trig_LK13:RS(SET: #58, RESET1: #60)
#62 ton_lk13:TON(IN: #61.Q1, PT: t)
#63 err_LK13 <= #62.Q
#64 EQ(adress_in_rs1, 22)
#65 AND(#64, err_true_rs1)
#66 EQ(adress_in_rs1, 22)
#67 AND(#66, err_false_rs1)
#68 trig_d4_2:RS(SET: #65, RESET1: #67)
#69 ton_d4_2:TON(IN: #68.Q1, PT: t)
#70 err_D4_mod2 <= #69.Q
#71 EQ(adress_in_rs2, 14)
#72 AND(#71, err_true_rs2)
#73 EQ(adress_in_rs2, 14)
#74 AND(#73, err_false_rs2)
#75 trig_gr3:RS(SET: #72, RESET1: #74)
#76 ton_gr3:TON(IN: #75.Q1, PT: t)
#77 err_GR3 <= #76.Q
#78 EQ(adress_in_rs1, 25)
#79 AND(#78, err_true_rs1)
#80 EQ(adress_in_rs1, 25)
#81 AND(#80, err_false_rs1)
#82 trig_d2:RS(SET: #79, RESET1: #81)
#83 ton_d2:TON(IN: #82.Q1, PT: t)
#84 err_D2 <= #83.Q
#85 EQ(adress_in_rs1, 7)
#86 AND(#85, err_true_rs1)
#87 EQ(adress_in_rs1, 7)
#88 AND(#87, err_false_rs1)
#89 trig_lk7:RS(SET: #86, RESET1: #88)
#90 ton_lk7:TON(IN: #89.Q1, PT: t)
#91 err_LK7 <= #90.Q
#92 EQ(adress_in_rs2, 26)
#93 AND(#92, err_true_rs2)
#94 EQ(adress_in_rs2, 26)
#95 AND(#94, err_false_rs2)
#96 trig_cyc:RS(SET: #93, RESET1: #95)
#97 ton_cyc:TON(IN: #96.Q1, PT: t)
#98 err_cyc1 <= #97.Q
#99 EQ(adress_in_rs1, 8)
#100 AND(#99, err_true_rs1)
#101 EQ(adress_in_rs1, 8)
#102 AND(#101, err_false_rs1)
#103 trig_lk8:RS(SET: #100, RESET1: #102)
#104 ton_lk8:TON(IN: #103.Q1, PT: t)
#105 err_LK8 <= #104.Q
#106 EQ(adress_in_rs2, 27)
#107 AND(#106, err_true_rs2)
#108 EQ(adress_in_rs2, 27)
#109 AND(#108, err_false_rs2)
#110 trig_cyc1:RS(SET: #107, RESET1: #109)
#111 ton_cyc1:TON(IN: #110.Q1, PT: t)
#112 err_cyc2 <= #111.Q
#113 EQ(adress_in_rs2, 6)
#114 AND(#113, err_true_rs2)
#115 EQ(adress_in_rs2, 6)
#116 AND(#115, err_false_rs2)
#117 trig_lk6:RS(SET: #114, RESET1: #116)
#118 ton_lk6:TON(IN: #117.Q1, PT: t)
#119 err_LK6 <= #118.Q
#120 EQ(adress_in_rs2, 9)
#121 AND(#120, err_true_rs2)
#122 EQ(adress_in_rs2, 9)
#123 AND(#122, err_false_rs2)
#124 trig_LK9:RS(SET: #121, RESET1: #123)
#125 ton_lk9:TON(IN: #124.Q1, PT: t)
#126 err_LK9 <= #125.Q
#127 EQ(adress_in_rs2, 18)
#128 AND(#127, err_true_rs2)
#129 EQ(adress_in_rs2, 18)
#130 AND(#129, err_false_rs2)
#131 trig_LP1_3_1:RS(SET: #128, RESET1: #130)
#132 ton_LP1_3_1:TON(IN: #131.Q1, PT: t)
#133 err_LP1_3_mod1 <= #132.Q
#134 EQ(adress_in_rs2, 19)
#135 AND(#134, err_true_rs2)
#136 EQ(adress_in_rs2, 19)
#137 AND(#136, err_false_rs2)
#138 trig_LP1_3_2:RS(SET: #135, RESET1: #137)
#139 ton_LP1_3_2:TON(IN: #138.Q1, PT: t)
#140 err_LP1_3_mod2 <= #139.Q
#141 EQ(adress_in_rs2, 15)
#142 AND(#141, err_true_rs2)
#143 EQ(adress_in_rs2, 15)
#144 AND(#143, err_false_rs2)
#145 trig_GR2:RS(SET: #142, RESET1: #144)
#146 ton_GR2:TON(IN: #145.Q1, PT: t)
#147 err_GR2 <= #146.Q
#148 EQ(adress_in_rs1, 5)
#149 AND(#148, err_true_rs1)
#150 EQ(adress_in_rs1, 5)
#151 AND(#150, err_false_rs1)
#152 trig_lk5:RS(SET: #149, RESET1: #151)
#153 ton_lk5:TON(IN: #152.Q1, PT: t)
#154 err_lk5 <= #153.Q
#155 EQ(adress_in_rs1, 16)
#156 AND(#155, err_true_rs1)
#157 EQ(adress_in_rs1, 16)
#158 AND(#157, err_false_rs1)
#159 trig_lp4:RS(SET: #156, RESET1: #158)
#160 ton_lp4:TON(IN: #159.Q1, PT: t)
#161 err_lp4 <= #160.Q
#162 EQ(adress_in_rs1, 17)
#163 AND(#162, err_true_rs1)
#164 EQ(adress_in_rs1, 17)
#165 AND(#164, err_false_rs1)
#166 trig_lp5:RS(SET: #163, RESET1: #165)
#167 ton_lp5:TON(IN: #166.Q1, PT: t)
#168 err_lp5 <= #167.Q
#169 EQ(adress_in_rs2, 4)
#170 AND(#169, err_true_rs2)
#171 EQ(adress_in_rs2, 4)
#172 AND(#171, err_false_rs2)
#173 trig_lk4:RS(SET: #170, RESET1: #172)
#174 ton_lk4:TON(IN: #173.Q1, PT: t)
#175 err_lk4 <= #174.Q
#176 EQ(adress_in_rs2, 1)
#177 AND(#176, err_true_rs2)
#178 EQ(adress_in_rs2, 1)
#179 AND(#178, err_false_rs2)
#180 trig_gr1:RS(SET: #177, RESET1: #179)
#181 ton_gr1:TON(IN: #180.Q1, PT: t)
#182 err_gr1 <= #181.Q
#183 EQ(adress_in_rs2, 2)
#184 AND(#183, err_true_rs2)
#185 EQ(adress_in_rs2, 2)
#186 AND(#185, err_false_rs2)
#187 trig_lk2:RS(SET: #184, RESET1: #186)
#188 ton_lk2:TON(IN: #187.Q1, PT: t)
#189 err_lk2 <= #188.Q
#190 EQ(adress_in_rs2, 3)
#191 AND(#190, err_true_rs2)
#192 EQ(adress_in_rs2, 3)
#193 AND(#192, err_false_rs2)
#194 trig_lk3:RS(SET: #191, RESET1: #193)
#195 ton_lk3:TON(IN: #194.Q1, PT: t)
#196 err_lk3 <= #195.Q
#197 EQ(adress_in_rs1, 1)
#198 AND(#197, err_true_rs1)
#199 EQ(adress_in_rs1, 1)
#200 AND(#199, err_false_rs1)
#201 trig_lp4_temp:RS(SET: #198, RESET1: #200)
#202 ton_lp4_temp:TON(IN: #201.Q1, PT: t)
#203 err_lp4_temp <= #202.Q
#204 EQ(adress_in_rs1, 2)
#205 AND(#204, err_true_rs1)
#206 EQ(adress_in_rs1, 2)
#207 AND(#206, err_false_rs1)
#208 trig_d3_temp:RS(SET: #205, RESET1: #207)
#209 ton_d3_temp:TON(IN: #208.Q1, PT: t)
#210 err_d3_temp <= #209.Q
#211 EQ(adress_in_rs1, 3)
#212 AND(#211, err_true_rs1)
#213 EQ(adress_in_rs1, 3)
#214 AND(#213, err_false_rs1)
#215 trig_d4_temp:RS(SET: #212, RESET1: #214)
#216 ton_d4_temp:TON(IN: #215.Q1, PT: t)
#217 err_d4_temp <= #216.Q
#218 EQ(adress_in_rs2, 44)
#219 AND(#218, err_true_rs1)
#220 EQ(adress_in_rs2, 44)
#221 AND(#220, err_false_rs1)
#222 trig_vp1_temp:RS(SET: #219, RESET1: #221)
#223 ton_vp1_temp:TON(IN: #222.Q1, PT: t)
#224 err_vp1_temp <= #223.Q
_END_CFC_
(* the same logic as Structured Text *)
(* Если есть ошибка на выходе true; нет - false *)
(* Если по определенному адресу есть ошибка, то на выходе, / через выдержку времени, устанавливается true *)
err_true_rs1 := error_81_in_rs1 = 81;
err_true_rs2 := error_81_in_rs2 = 81;
err_false_rs1 := error_81_in_rs1 = 0;
err_false_rs2 := error_81_in_rs2 = 0;
trig_vp1(SET := (adress_in_rs2 = 20) AND err_true_rs2, RESET1 := (adress_in_rs2 = 20) AND err_false_rs2);
ton_vp1(IN := trig_vp1.Q1, PT := t);
err_vp1 := ton_vp1.Q;
trig_LK10(SET := (adress_in_rs2 = 10) AND err_true_rs2, RESET1 := (adress_in_rs2 = 10) AND err_false_rs2);
ton_lk10(IN := trig_LK10.Q1, PT := t);
err_LK10 := ton_lk10.Q;
trig_d3_1(SET := (adress_in_rs1 = 24) AND err_true_rs1, RESET1 := (adress_in_rs1 = 24) AND err_false_rs1);
ton_d3_1(IN := trig_d3_1.Q1, PT := t);
err_D3_mod1 := ton_d3_1.Q;
trig_LK11(SET := (adress_in_rs2 = 11) AND err_true_rs2, RESET1 := (adress_in_rs2 = 11) AND err_false_rs2);
ton_lk11(IN := trig_LK11.Q1, PT := t);
err_LK11 := ton_lk11.Q;
trig_d3_2(SET := (adress_in_rs1 = 23) AND err_true_rs1, RESET1 := (adress_in_rs1 = 23) AND err_false_rs1);
ton_d3_2(IN := trig_d3_2.Q1, PT := t);
err_D3_mod2 := ton_d3_2.Q;
trig_LK12(SET := (adress_in_rs2 = 12) AND err_true_rs2, RESET1 := (adress_in_rs2 = 12) AND err_false_rs2);
ton_lk12(IN := trig_LK12.Q1, PT := t);
err_LK12 := ton_lk12.Q;
trig_d4_1(SET := (adress_in_rs1 = 21) AND err_true_rs1, RESET1 := (adress_in_rs1 = 21) AND err_false_rs1);
ton_d4_1(IN := trig_d4_1.Q1, PT := t);
err_D4_mod1 := ton_d4_1.Q;
trig_LK13(SET := (adress_in_rs2 = 13) AND err_true_rs2, RESET1 := (adress_in_rs2 = 13) AND err_false_rs2);
ton_lk13(IN := trig_LK13.Q1, PT := t);
err_LK13 := ton_lk13.Q;
trig_d4_2(SET := (adress_in_rs1 = 22) AND err_true_rs1, RESET1 := (adress_in_rs1 = 22) AND err_false_rs1);
ton_d4_2(IN := trig_d4_2.Q1, PT := t);
err_D4_mod2 := ton_d4_2.Q;
trig_gr3(SET := (adress_in_rs2 = 14) AND err_true_rs2, RESET1 := (adress_in_rs2 = 14) AND err_false_rs2);
ton_gr3(IN := trig_gr3.Q1, PT := t);
err_GR3 := ton_gr3.Q;
trig_d2(SET := (adress_in_rs1 = 25) AND err_true_rs1, RESET1 := (adress_in_rs1 = 25) AND err_false_rs1);
ton_d2(IN := trig_d2.Q1, PT := t);
err_D2 := ton_d2.Q;
trig_lk7(SET := (adress_in_rs1 = 7) AND err_true_rs1, RESET1 := (adress_in_rs1 = 7) AND err_false_rs1);
ton_lk7(IN := trig_lk7.Q1, PT := t);
err_LK7 := ton_lk7.Q;
trig_cyc(SET := (adress_in_rs2 = 26) AND err_true_rs2, RESET1 := (adress_in_rs2 = 26) AND err_false_rs2);
ton_cyc(IN := trig_cyc.Q1, PT := t);
err_cyc1 := ton_cyc.Q;
trig_lk8(SET := (adress_in_rs1 = 8) AND err_true_rs1, RESET1 := (adress_in_rs1 = 8) AND err_false_rs1);
ton_lk8(IN := trig_lk8.Q1, PT := t);
err_LK8 := ton_lk8.Q;
trig_cyc1(SET := (adress_in_rs2 = 27) AND err_true_rs2, RESET1 := (adress_in_rs2 = 27) AND err_false_rs2);
ton_cyc1(IN := trig_cyc1.Q1, PT := t);
err_cyc2 := ton_cyc1.Q;
trig_lk6(SET := (adress_in_rs2 = 6) AND err_true_rs2, RESET1 := (adress_in_rs2 = 6) AND err_false_rs2);
ton_lk6(IN := trig_lk6.Q1, PT := t);
err_LK6 := ton_lk6.Q;
trig_LK9(SET := (adress_in_rs2 = 9) AND err_true_rs2, RESET1 := (adress_in_rs2 = 9) AND err_false_rs2);
ton_lk9(IN := trig_LK9.Q1, PT := t);
err_LK9 := ton_lk9.Q;
trig_LP1_3_1(SET := (adress_in_rs2 = 18) AND err_true_rs2, RESET1 := (adress_in_rs2 = 18) AND err_false_rs2);
ton_LP1_3_1(IN := trig_LP1_3_1.Q1, PT := t);
err_LP1_3_mod1 := ton_LP1_3_1.Q;
trig_LP1_3_2(SET := (adress_in_rs2 = 19) AND err_true_rs2, RESET1 := (adress_in_rs2 = 19) AND err_false_rs2);
ton_LP1_3_2(IN := trig_LP1_3_2.Q1, PT := t);
err_LP1_3_mod2 := ton_LP1_3_2.Q;
trig_GR2(SET := (adress_in_rs2 = 15) AND err_true_rs2, RESET1 := (adress_in_rs2 = 15) AND err_false_rs2);
ton_GR2(IN := trig_GR2.Q1, PT := t);
err_GR2 := ton_GR2.Q;
trig_lk5(SET := (adress_in_rs1 = 5) AND err_true_rs1, RESET1 := (adress_in_rs1 = 5) AND err_false_rs1);
ton_lk5(IN := trig_lk5.Q1, PT := t);
err_lk5 := ton_lk5.Q;
trig_lp4(SET := (adress_in_rs1 = 16) AND err_true_rs1, RESET1 := (adress_in_rs1 = 16) AND err_false_rs1);
ton_lp4(IN := trig_lp4.Q1, PT := t);
err_lp4 := ton_lp4.Q;
trig_lp5(SET := (adress_in_rs1 = 17) AND err_true_rs1, RESET1 := (adress_in_rs1 = 17) AND err_false_rs1);
ton_lp5(IN := trig_lp5.Q1, PT := t);
err_lp5 := ton_lp5.Q;
trig_lk4(SET := (adress_in_rs2 = 4) AND err_true_rs2, RESET1 := (adress_in_rs2 = 4) AND err_false_rs2);
ton_lk4(IN := trig_lk4.Q1, PT := t);
err_lk4 := ton_lk4.Q;
trig_gr1(SET := (adress_in_rs2 = 1) AND err_true_rs2, RESET1 := (adress_in_rs2 = 1) AND err_false_rs2);
ton_gr1(IN := trig_gr1.Q1, PT := t);
err_gr1 := ton_gr1.Q;
trig_lk2(SET := (adress_in_rs2 = 2) AND err_true_rs2, RESET1 := (adress_in_rs2 = 2) AND err_false_rs2);
ton_lk2(IN := trig_lk2.Q1, PT := t);
err_lk2 := ton_lk2.Q;
trig_lk3(SET := (adress_in_rs2 = 3) AND err_true_rs2, RESET1 := (adress_in_rs2 = 3) AND err_false_rs2);
ton_lk3(IN := trig_lk3.Q1, PT := t);
err_lk3 := ton_lk3.Q;
trig_lp4_temp(SET := (adress_in_rs1 = 1) AND err_true_rs1, RESET1 := (adress_in_rs1 = 1) AND err_false_rs1);
ton_lp4_temp(IN := trig_lp4_temp.Q1, PT := t);
err_lp4_temp := ton_lp4_temp.Q;
trig_d3_temp(SET := (adress_in_rs1 = 2) AND err_true_rs1, RESET1 := (adress_in_rs1 = 2) AND err_false_rs1);
ton_d3_temp(IN := trig_d3_temp.Q1, PT := t);
err_d3_temp := ton_d3_temp.Q;
trig_d4_temp(SET := (adress_in_rs1 = 3) AND err_true_rs1, RESET1 := (adress_in_rs1 = 3) AND err_false_rs1);
ton_d4_temp(IN := trig_d4_temp.Q1, PT := t);
err_d4_temp := ton_d4_temp.Q;
trig_vp1_temp(SET := (adress_in_rs2 = 44) AND err_true_rs1, RESET1 := (adress_in_rs2 = 44) AND err_false_rs1);
ton_vp1_temp(IN := trig_vp1_temp.Q1, PT := t);
err_vp1_temp := ton_vp1_temp.Q;
END_FUNCTION_BLOCK

(* POU if_Hz, ST *)
FUNCTION_BLOCK if_Hz (*блок установки входящей частоты для частотника -
						если введенная частота ниже 20Гц аатоматически установить 20Гц, если выше 50Гц - установить 50Гц*)
VAR_INPUT
	input_Hz_LP4_if: WORD;
	input_Hz_LP5_if: WORD;
END_VAR
VAR_OUTPUT
	output_Hz_LP4_if: WORD;
	output_Hz_LP5_if: WORD;
END_VAR
VAR
END_VAR
IF input_Hz_LP4_if < 20
THEN output_Hz_LP4_if := 45;
ELSE output_Hz_LP4_if := input_Hz_LP4_if;
END_IF;

IF input_Hz_LP4_if >= 50
THEN output_Hz_LP4_if := 50;
END_IF;

IF input_Hz_LP5_if < 20
THEN output_Hz_LP5_if := 45;
ELSE output_Hz_LP5_if := input_Hz_LP5_if;
END_IF;

IF input_Hz_LP5_if >= 50
THEN output_Hz_LP5_if := 50;
END_IF;
END_FUNCTION_BLOCK

(* POU PP1, LD *)
FUNCTION_BLOCK PP1
VAR_INPUT
	P_LK2_in: BOOL;
	stop_pp_LK3: BOOL;
	LV2: BOOL;
	LV1: BOOL;
	pusk_s:BOOL;
	stop_s: BOOL;
END_VAR
VAR_OUTPUT
	KM1_PP1: BOOL;
END_VAR
VAR
	stop_pp1: BOOL;
	high_GR1: BOOL;
	sr_GR1: SR;
	stop_pp: R_TRIG;
	sr_pp: SR;
END_VAR
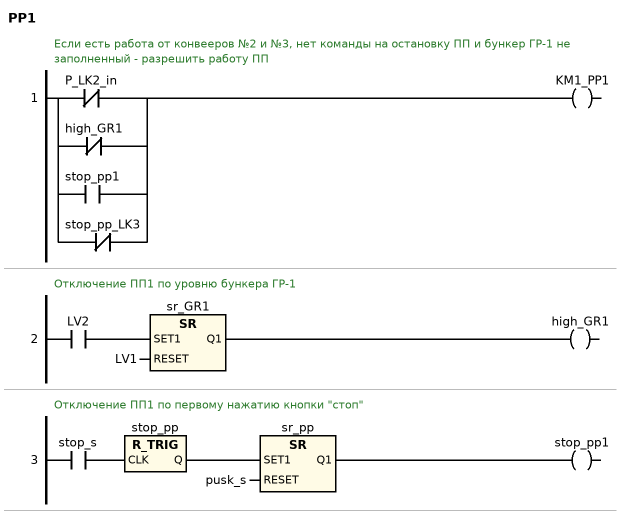
_LD_ (* Ladder Diagram *)
NETWORK 1 (* Если есть работа от конвееров №2 и №3, нет команды на остановку ПП и бункер ГР-1 не заполненный - разрешить работу ПП *)
	{ [/P_LK2_in] | [/high_GR1] | [stop_pp1] | [/stop_pp_LK3] } --- (KM1_PP1)
NETWORK 2 (* Отключение ПП1 по уровню бункера ГР-1 *)
	[LV2] - sr_GR1:SR(SET1: *, RESET: LV1) --- (high_GR1)
NETWORK 3 (* Отключение ПП1 по первому нажатию кнопки "стоп" *)
	[stop_s] - stop_pp:R_TRIG(CLK: *) - sr_pp:SR(SET1: *, RESET: pusk_s) --- (stop_pp1)
_END_LD_
(* the same logic as Structured Text *)
(* Network 1: Если есть работа от конвееров №2 и №3, нет команды на остановку ПП и бункер ГР-1 не заполненный - разрешить работу ПП *)
KM1_PP1 := NOT P_LK2_in OR NOT high_GR1 OR stop_pp1 OR NOT stop_pp_LK3;
(* Network 2: Отключение ПП1 по уровню бункера ГР-1 *)
sr_GR1(SET1 := LV2, RESET := LV1);
high_GR1 := sr_GR1.Q1;
(* Network 3: Отключение ПП1 по первому нажатию кнопки "стоп" *)
stop_pp(CLK := stop_s);
sr_pp(SET1 := stop_pp.Q, RESET := pusk_s);
stop_pp1 := sr_pp.Q1;
END_FUNCTION_BLOCK

(* POU bool_to, CFC *)
FUNCTION_BLOCK bool_to (* блок преобразования word-значений из сети в bool-значения, для управляющих сигналов*)
VAR_INPUT
	pusk_LAN_LP4: WORD;
	stop_LAN_LP4: WORD;
	pusk_LAN_LP5: WORD;
	stop_LAN_LP5: WORD;
	pusk_LAN_VP1: WORD;
	stop_LAN_VP1: WORD;
	pusk_lan_LK10: WORD;
	pusk_lan_LK11: WORD;
	pusk_lan_LK12: WORD;
	pusk_lan_LK13: WORD;
	pusk_lan_GR3: WORD;
	pusk_lan_LK7: WORD;
	pusk_lan_LK8: WORD;
	pusk_lan_LK6: WORD;
	pusk_lan_LK9: WORD;
	pusk_lan_LP1_3: WORD;
	pusk_lan_GR2: WORD;
	pusk_lan_LK5: WORD;
	pusk_lan_LK4: WORD;
	pusk_lan_LK3: WORD;
	pusk_lan_GR1: WORD;
	pusk_lan_LK2: WORD;
	stop_lan_LK10: WORD;
	stop_lan_LK11: WORD;
	stop_lan_LK12: WORD;
	stop_lan_LK13: WORD;
	stop_lan_GR3: WORD;
	stop_lan_LK7: WORD;
	stop_lan_LK8: WORD;
	stop_lan_LK6: WORD;
	stop_lan_LK9: WORD;
	stop_lan_LP1_3: WORD;
	stop_lan_GR2: WORD;
	stop_lan_LK5: WORD;
	stop_lan_LK4: WORD;
	stop_lan_LK3: WORD;
	stop_lan_GR1: WORD;
	stop_lan_LK2: WORD;
	stop_LAN_D3: WORD;
	stop_LAN_D4: WORD;
	pusk_lan_D2: WORD;
	stop_lan_D2: WORD;
	pusk_lan_D3: WORD;
	pusk_lan_D4: WORD;
	pusk_lan_cyclone: WORD;
	stop_lan_cyclone: WORD;
	tros_self_lk10_in: WORD;
	shod_self_lk10_in: WORD;
	ogr_self_lk10_in: WORD;
	vl_self_lk10_in: WORD;
	tros_self_lk11_in: WORD;
	shod_self_lk11_in: WORD;
	ogr_self_lk11_in: WORD;
	vl_self_lk11_in: WORD;
	tros_self_lk12_in: WORD;
	shod_self_lk12_in: WORD;
	ogr_self_lk12_in: WORD;
	vl_self_lk12_in: WORD;
	tros_self_lk13_in: WORD;
	shod_self_lk13_in: WORD;
	ogr_self_lk13_in: WORD;
	vl_self_lk13_in: WORD;
	tros_self_lk7_in: WORD;
	shod_self_lk7_in: WORD;
	ogr_self_lk7_in: WORD;
	vl_self_lk7_in: WORD;
	tros_self_lk8_in: WORD;
	shod_self_lk8_in: WORD;
	ogr_self_lk8_in: WORD;
	vl_self_lk8_in: WORD;
	tros_self_lk6_in: WORD;
	shod_self_lk6_in: WORD;
	ogr_self_lk6_in: WORD;
	vl_self_lk6_in: WORD;
	tros_self_lk9_in: WORD;
	shod_self_lk9_in: WORD;
	ogr_self_lk9_in: WORD;
	vl_self_lk9_in: WORD;
	vl_self_lp1_3_in: WORD;
	tros_self_lk5_in: WORD;
	shod_self_lk5_in: WORD;
	ogr_self_lk5_in: WORD;
	vl_self_lk5_in: WORD;
	tros_self_lk4_in: WORD;
	shod_self_lk4_in: WORD;
	vl_self_lk4_in: WORD;
	tros_self_lk3_in: WORD;
	shod_self_lk3_in: WORD;
	ogr_self_lk3_in: WORD;
	vl_self_lk3_in: WORD;
	tros_self_lk2_in: WORD;
	shod_self_lk2_in: WORD;
	ogr_self_lk2_in: WORD;
	vl_self_lk2_in: WORD;
	revers_in: WORD;
	vl_self_lp4_in: WORD;
	vl_self_lp5_in: WORD;
	pusk_shnek_razg_in: WORD;
	stop_shnek_razg_in: WORD;
	pusk_cyc_cleen_in: WORD;
	stop_cyc_cleen_in: WORD;
END_VAR
VAR_OUTPUT
	pusk_LAN_LP4_out: BOOL;
	stop_LAN_LP4_out: BOOL;
	pusk_LAN_LP5_out: BOOL;
	stop_LAN_LP5_out: BOOL;
	pusk_LAN_VP1_out: BOOL;
	stop_LAN_VP1_out: BOOL;
	pusk_lan_LK10_out: BOOL;
	pusk_lan_LK11_out: BOOL;
	pusk_lan_LK12_out: BOOL;
	pusk_lan_LK13_out: BOOL;
	pusk_lan_GR3_out: BOOL;
	pusk_lan_LK7out: BOOL;
	pusk_lan_LK8_out: BOOL;
	pusk_lan_LK6_out: BOOL;
	pusk_lan_LK9_out: BOOL;
	pusk_lan_LP1_3_out: BOOL;
	pusk_lan_GR2_out: BOOL;
	pusk_lan_LK5_out: BOOL;
	pusk_lan_LK4_out: BOOL;
	pusk_lan_LK3_out: BOOL;
	pusk_lan_GR1_out: BOOL;
	pusk_lan_LK2_out: BOOL;
	stop_lan_LK10_out: BOOL;
	stop_lan_LK11_out: BOOL;
	stop_lan_LK12_out: BOOL;
	stop_lan_LK13_out: BOOL;
	stop_lan_GR3_out: BOOL;
	stop_lan_LK7_out: BOOL;
	stop_lan_LK8_out: BOOL;
	stop_lan_LK6_out: BOOL;
	stop_lan_LK9_out: BOOL;
	stop_lan_LP1_3_out: BOOL;
	stop_lan_GR2_out: BOOL;
	stop_lan_LK5_out: BOOL;
	stop_lan_LK4_out: BOOL;
	stop_lan_LK3_out: BOOL;
	stop_lan_GR1_out: BOOL;
	stop_lan_LK2_out: BOOL;
	stop_LAN_D3_out: BOOL;
	stop_LAN_D4_out: BOOL;
	pusk_lan_D2_out: BOOL;
	stop_lan_D2_out: BOOL;
	pusk_lan_D3_out: BOOL;
	pusk_lan_D4_out: BOOL;
	pusk_lan_cyclone_out: BOOL;
	stop_lan_cyclone_out: BOOL;
	tros_self_lk10_out: BOOL;
	shod_self_lk10_out: BOOL;
	ogr_self_lk10_out: BOOL;
	vl_self_lk10_out: BOOL;
	tros_self_lk11_out: BOOL;
	shod_self_lk11_out: BOOL;
	ogr_self_lk11_out: BOOL;
	vl_self_lk11_out: BOOL;
	tros_self_lk12_out: BOOL;
	shod_self_lk12_out: BOOL;
	ogr_self_lk12_out: BOOL;
	vl_self_lk12_out: BOOL;
	tros_self_lk13_out: BOOL;
	shod_self_lk13_out: BOOL;
	ogr_self_lk13_out: BOOL;
	vl_self_lk13_out: BOOL;
	tros_self_lk7_out: BOOL;
	shod_self_lk7_out: BOOL;
	ogr_self_lk7_out: BOOL;
	vl_self_lk7_out: BOOL;
	tros_self_lk8_out: BOOL;
	shod_self_lk8_out: BOOL;
	ogr_self_lk8_out: BOOL;
	vl_self_lk8_out: BOOL;
	tros_self_lk6_out: BOOL;
	shod_self_lk6_out: BOOL;
	ogr_self_lk6_out: BOOL;
	vl_self_lk6_out: BOOL;
	tros_self_lk9_out: BOOL;
	shod_self_lk9_out: BOOL;
	ogr_self_lk9_out: BOOL;
	vl_self_lk9_out: BOOL;
	vl_self_lp1_3_out: BOOL;
	tros_self_lk5_out: BOOL;
	shod_self_lk5_out: BOOL;
	ogr_self_lk5_out: BOOL;
	vl_self_lk5_out: BOOL;
	tros_self_lk4_out: BOOL;
	shod_self_lk4_out: BOOL;
	vl_self_lk4_out: BOOL;
	tros_self_lk3_out: BOOL;
	shod_self_lk3_out: BOOL;
	ogr_self_lk3_out: BOOL;
	vl_self_lk3_out: BOOL;
	tros_self_lk2_out: BOOL;
	shod_self_lk2_out: BOOL;
	ogr_self_lk2_out: BOOL;
	vl_self_lk2_out: BOOL;
	revers_out: BOOL;
	vl_self_lp4_out: BOOL;
	vl_self_lp5_out: BOOL;
	pusk_shnek_razg_out: BOOL;
	stop_shnek_razg_out: BOOL;
	pusk_cyc_cleen_out: BOOL;
	stop_cyc_cleen_out: BOOL;
END_VAR
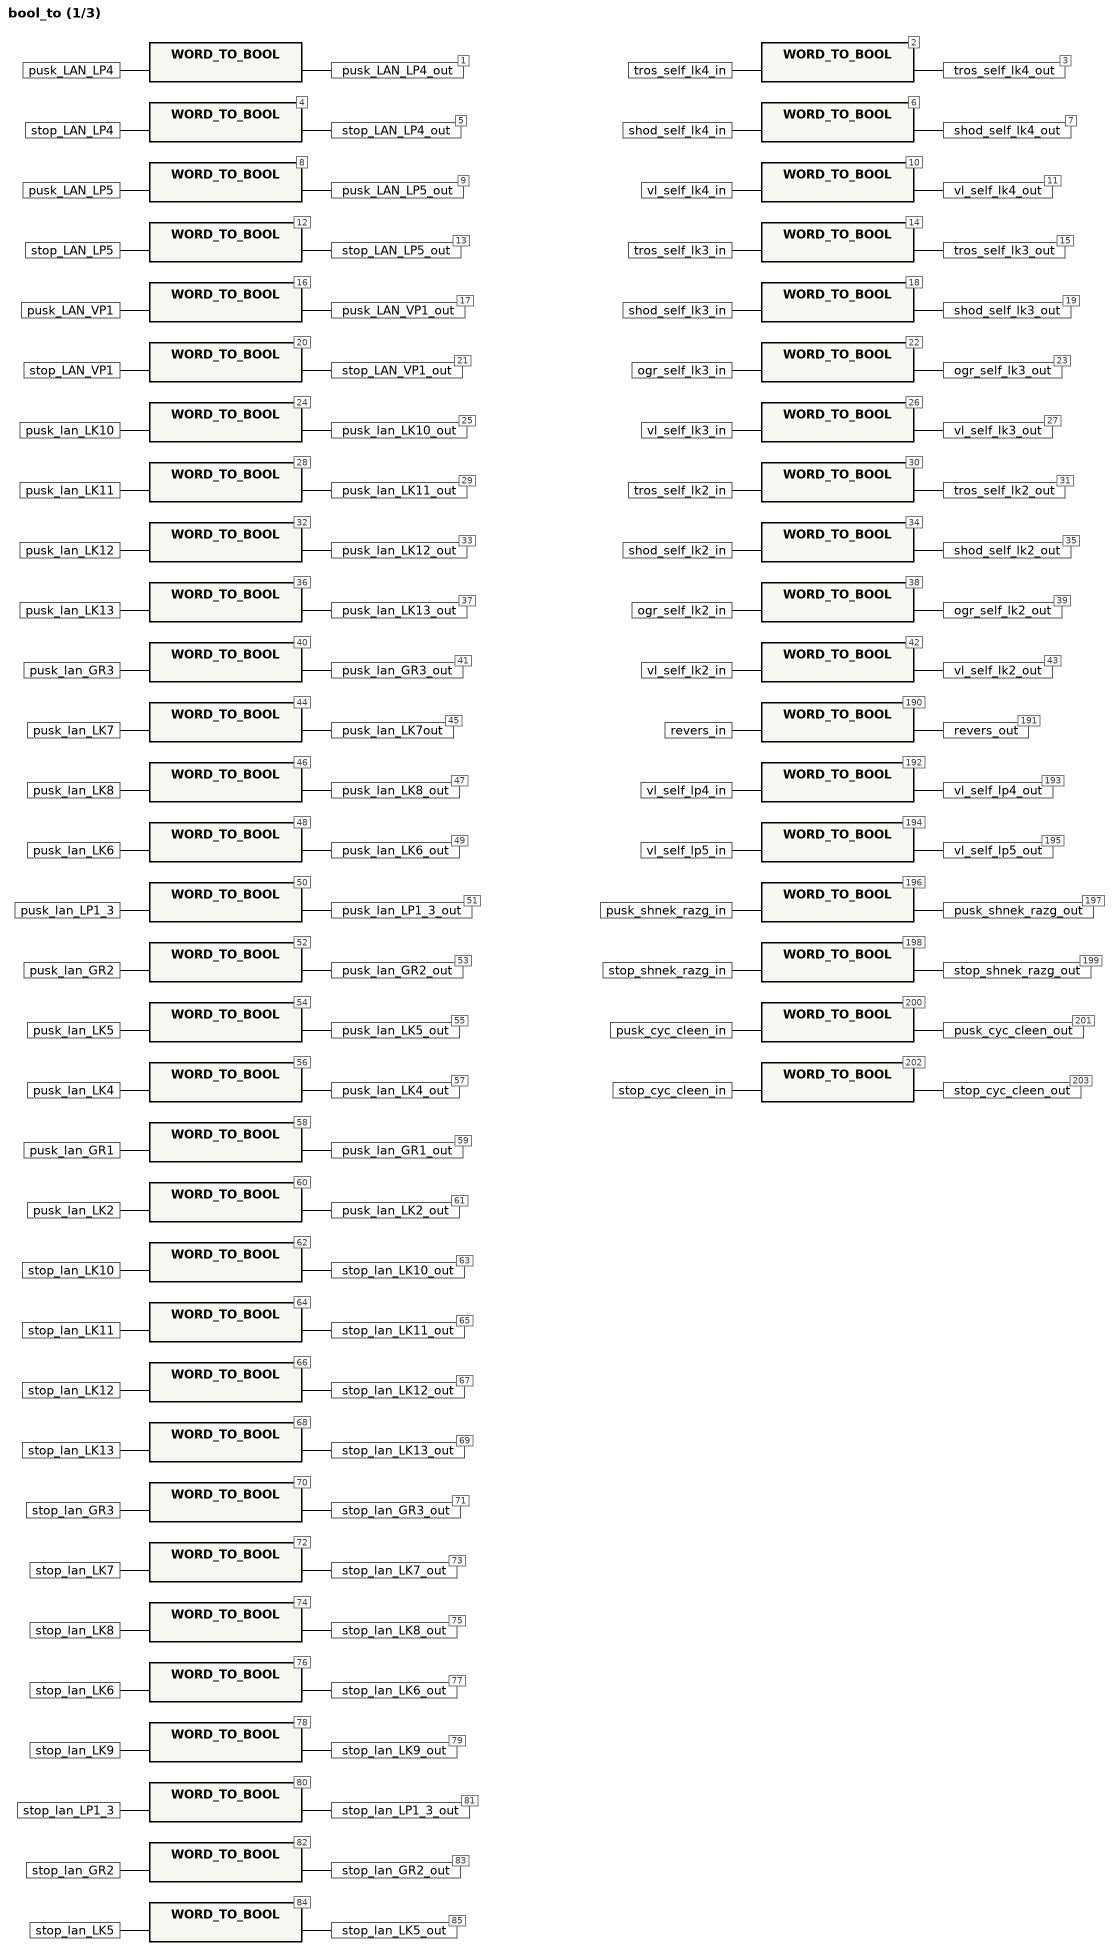
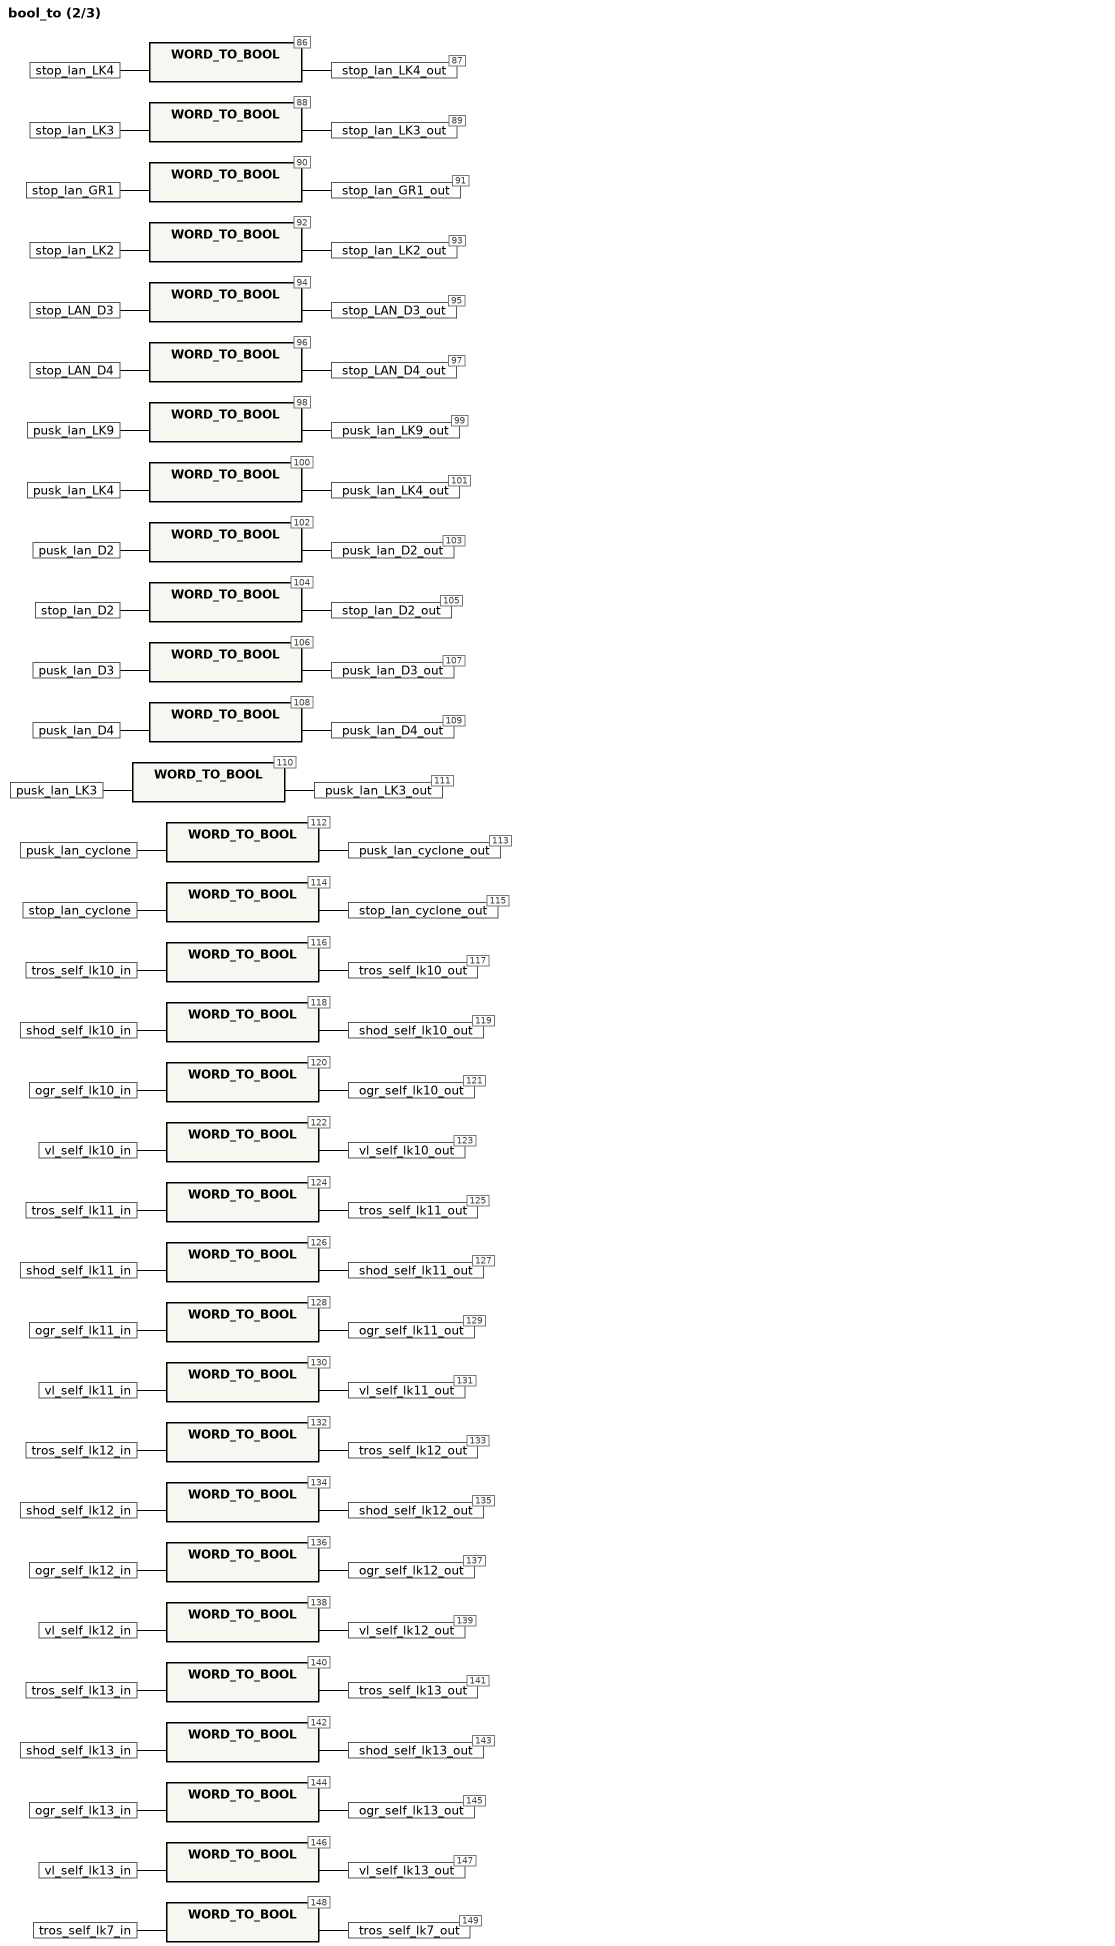
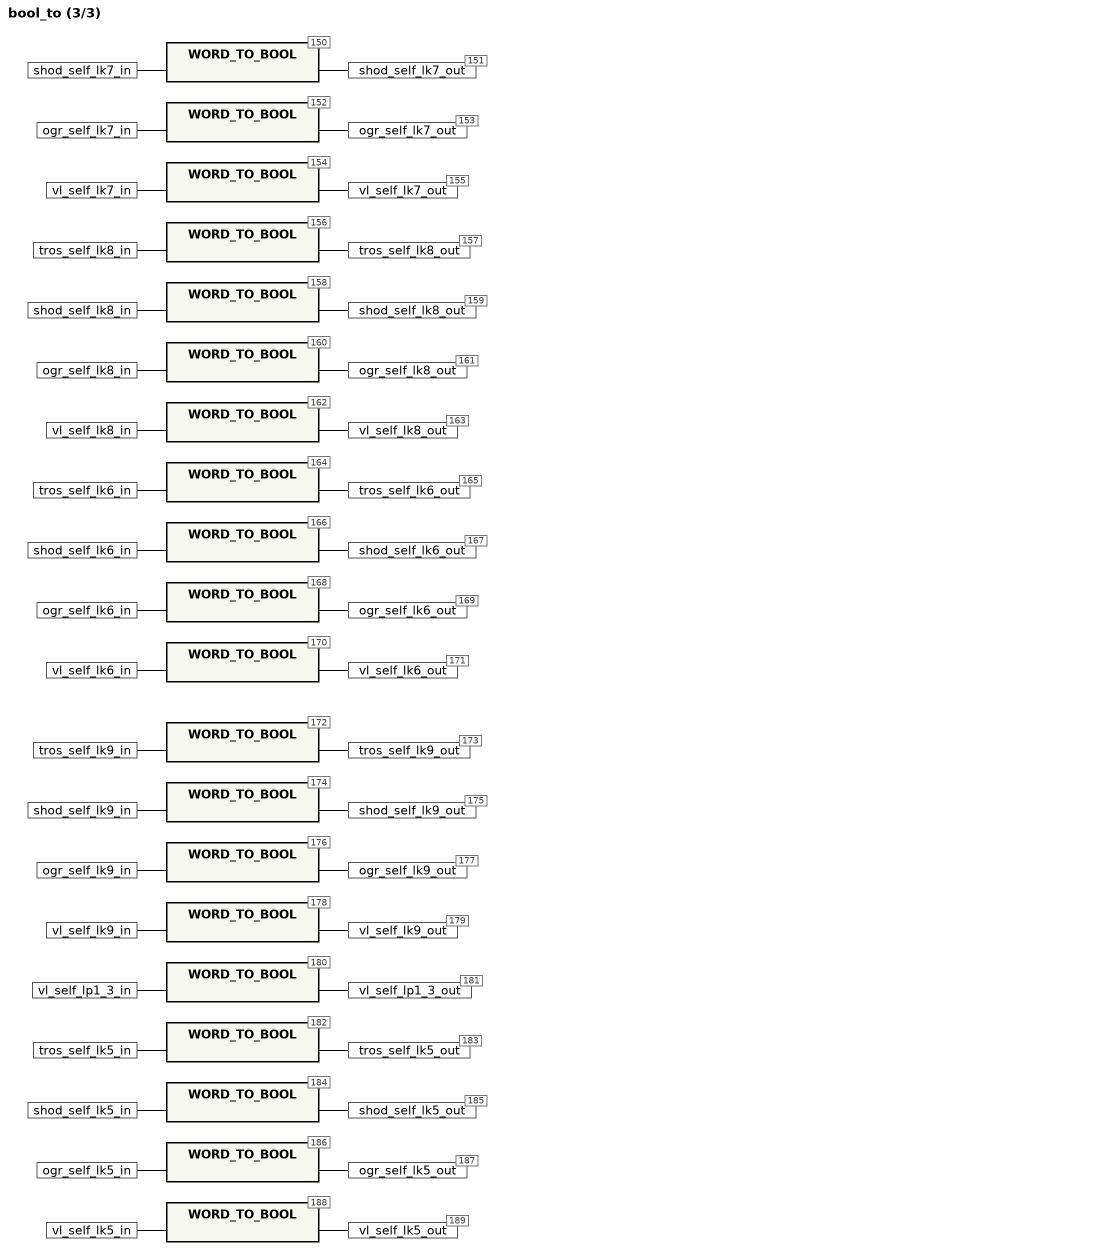
_CFC_ (* Continuous Function Chart, elements in execution order *)
#0 WORD_TO_BOOL(pusk_LAN_LP4)
#1 pusk_LAN_LP4_out <= #0
#2 WORD_TO_BOOL(tros_self_lk4_in)
#3 tros_self_lk4_out <= #2
#4 WORD_TO_BOOL(stop_LAN_LP4)
#5 stop_LAN_LP4_out <= #4
#6 WORD_TO_BOOL(shod_self_lk4_in)
#7 shod_self_lk4_out <= #6
#8 WORD_TO_BOOL(pusk_LAN_LP5)
#9 pusk_LAN_LP5_out <= #8
#10 WORD_TO_BOOL(vl_self_lk4_in)
#11 vl_self_lk4_out <= #10
#12 WORD_TO_BOOL(stop_LAN_LP5)
#13 stop_LAN_LP5_out <= #12
#14 WORD_TO_BOOL(tros_self_lk3_in)
#15 tros_self_lk3_out <= #14
#16 WORD_TO_BOOL(pusk_LAN_VP1)
#17 pusk_LAN_VP1_out <= #16
#18 WORD_TO_BOOL(shod_self_lk3_in)
#19 shod_self_lk3_out <= #18
#20 WORD_TO_BOOL(stop_LAN_VP1)
#21 stop_LAN_VP1_out <= #20
#22 WORD_TO_BOOL(ogr_self_lk3_in)
#23 ogr_self_lk3_out <= #22
#24 WORD_TO_BOOL(pusk_lan_LK10)
#25 pusk_lan_LK10_out <= #24
#26 WORD_TO_BOOL(vl_self_lk3_in)
#27 vl_self_lk3_out <= #26
#28 WORD_TO_BOOL(pusk_lan_LK11)
#29 pusk_lan_LK11_out <= #28
#30 WORD_TO_BOOL(tros_self_lk2_in)
#31 tros_self_lk2_out <= #30
#32 WORD_TO_BOOL(pusk_lan_LK12)
#33 pusk_lan_LK12_out <= #32
#34 WORD_TO_BOOL(shod_self_lk2_in)
#35 shod_self_lk2_out <= #34
#36 WORD_TO_BOOL(pusk_lan_LK13)
#37 pusk_lan_LK13_out <= #36
#38 WORD_TO_BOOL(ogr_self_lk2_in)
#39 ogr_self_lk2_out <= #38
#40 WORD_TO_BOOL(pusk_lan_GR3)
#41 pusk_lan_GR3_out <= #40
#42 WORD_TO_BOOL(vl_self_lk2_in)
#43 vl_self_lk2_out <= #42
#44 WORD_TO_BOOL(pusk_lan_LK7)
#45 pusk_lan_LK7out <= #44
#46 WORD_TO_BOOL(pusk_lan_LK8)
#47 pusk_lan_LK8_out <= #46
#48 WORD_TO_BOOL(pusk_lan_LK6)
#49 pusk_lan_LK6_out <= #48
#50 WORD_TO_BOOL(pusk_lan_LP1_3)
#51 pusk_lan_LP1_3_out <= #50
#52 WORD_TO_BOOL(pusk_lan_GR2)
#53 pusk_lan_GR2_out <= #52
#54 WORD_TO_BOOL(pusk_lan_LK5)
#55 pusk_lan_LK5_out <= #54
#56 WORD_TO_BOOL(pusk_lan_LK4)
#57 pusk_lan_LK4_out <= #56
#58 WORD_TO_BOOL(pusk_lan_GR1)
#59 pusk_lan_GR1_out <= #58
#60 WORD_TO_BOOL(pusk_lan_LK2)
#61 pusk_lan_LK2_out <= #60
#62 WORD_TO_BOOL(stop_lan_LK10)
#63 stop_lan_LK10_out <= #62
#64 WORD_TO_BOOL(stop_lan_LK11)
#65 stop_lan_LK11_out <= #64
#66 WORD_TO_BOOL(stop_lan_LK12)
#67 stop_lan_LK12_out <= #66
#68 WORD_TO_BOOL(stop_lan_LK13)
#69 stop_lan_LK13_out <= #68
#70 WORD_TO_BOOL(stop_lan_GR3)
#71 stop_lan_GR3_out <= #70
#72 WORD_TO_BOOL(stop_lan_LK7)
#73 stop_lan_LK7_out <= #72
#74 WORD_TO_BOOL(stop_lan_LK8)
#75 stop_lan_LK8_out <= #74
#76 WORD_TO_BOOL(stop_lan_LK6)
#77 stop_lan_LK6_out <= #76
#78 WORD_TO_BOOL(stop_lan_LK9)
#79 stop_lan_LK9_out <= #78
#80 WORD_TO_BOOL(stop_lan_LP1_3)
#81 stop_lan_LP1_3_out <= #80
#82 WORD_TO_BOOL(stop_lan_GR2)
#83 stop_lan_GR2_out <= #82
#84 WORD_TO_BOOL(stop_lan_LK5)
#85 stop_lan_LK5_out <= #84
#86 WORD_TO_BOOL(stop_lan_LK4)
#87 stop_lan_LK4_out <= #86
#88 WORD_TO_BOOL(stop_lan_LK3)
#89 stop_lan_LK3_out <= #88
#90 WORD_TO_BOOL(stop_lan_GR1)
#91 stop_lan_GR1_out <= #90
#92 WORD_TO_BOOL(stop_lan_LK2)
#93 stop_lan_LK2_out <= #92
#94 WORD_TO_BOOL(stop_LAN_D3)
#95 stop_LAN_D3_out <= #94
#96 WORD_TO_BOOL(stop_LAN_D4)
#97 stop_LAN_D4_out <= #96
#98 WORD_TO_BOOL(pusk_lan_LK9)
#99 pusk_lan_LK9_out <= #98
#100 WORD_TO_BOOL(pusk_lan_LK4)
#101 pusk_lan_LK4_out <= #100
#102 WORD_TO_BOOL(pusk_lan_D2)
#103 pusk_lan_D2_out <= #102
#104 WORD_TO_BOOL(stop_lan_D2)
#105 stop_lan_D2_out <= #104
#106 WORD_TO_BOOL(pusk_lan_D3)
#107 pusk_lan_D3_out <= #106
#108 WORD_TO_BOOL(pusk_lan_D4)
#109 pusk_lan_D4_out <= #108
#110 WORD_TO_BOOL(pusk_lan_LK3)
#111 pusk_lan_LK3_out <= #110
#112 WORD_TO_BOOL(pusk_lan_cyclone)
#113 pusk_lan_cyclone_out <= #112
#114 WORD_TO_BOOL(stop_lan_cyclone)
#115 stop_lan_cyclone_out <= #114
#116 WORD_TO_BOOL(tros_self_lk10_in)
#117 tros_self_lk10_out <= #116
#118 WORD_TO_BOOL(shod_self_lk10_in)
#119 shod_self_lk10_out <= #118
#120 WORD_TO_BOOL(ogr_self_lk10_in)
#121 ogr_self_lk10_out <= #120
#122 WORD_TO_BOOL(vl_self_lk10_in)
#123 vl_self_lk10_out <= #122
#124 WORD_TO_BOOL(tros_self_lk11_in)
#125 tros_self_lk11_out <= #124
#126 WORD_TO_BOOL(shod_self_lk11_in)
#127 shod_self_lk11_out <= #126
#128 WORD_TO_BOOL(ogr_self_lk11_in)
#129 ogr_self_lk11_out <= #128
#130 WORD_TO_BOOL(vl_self_lk11_in)
#131 vl_self_lk11_out <= #130
#132 WORD_TO_BOOL(tros_self_lk12_in)
#133 tros_self_lk12_out <= #132
#134 WORD_TO_BOOL(shod_self_lk12_in)
#135 shod_self_lk12_out <= #134
#136 WORD_TO_BOOL(ogr_self_lk12_in)
#137 ogr_self_lk12_out <= #136
#138 WORD_TO_BOOL(vl_self_lk12_in)
#139 vl_self_lk12_out <= #138
#140 WORD_TO_BOOL(tros_self_lk13_in)
#141 tros_self_lk13_out <= #140
#142 WORD_TO_BOOL(shod_self_lk13_in)
#143 shod_self_lk13_out <= #142
#144 WORD_TO_BOOL(ogr_self_lk13_in)
#145 ogr_self_lk13_out <= #144
#146 WORD_TO_BOOL(vl_self_lk13_in)
#147 vl_self_lk13_out <= #146
#148 WORD_TO_BOOL(tros_self_lk7_in)
#149 tros_self_lk7_out <= #148
#150 WORD_TO_BOOL(shod_self_lk7_in)
#151 shod_self_lk7_out <= #150
#152 WORD_TO_BOOL(ogr_self_lk7_in)
#153 ogr_self_lk7_out <= #152
#154 WORD_TO_BOOL(vl_self_lk7_in)
#155 vl_self_lk7_out <= #154
#156 WORD_TO_BOOL(tros_self_lk8_in)
#157 tros_self_lk8_out <= #156
#158 WORD_TO_BOOL(shod_self_lk8_in)
#159 shod_self_lk8_out <= #158
#160 WORD_TO_BOOL(ogr_self_lk8_in)
#161 ogr_self_lk8_out <= #160
#162 WORD_TO_BOOL(vl_self_lk8_in)
#163 vl_self_lk8_out <= #162
#164 WORD_TO_BOOL(tros_self_lk6_in)
#165 tros_self_lk6_out <= #164
#166 WORD_TO_BOOL(shod_self_lk6_in)
#167 shod_self_lk6_out <= #166
#168 WORD_TO_BOOL(ogr_self_lk6_in)
#169 ogr_self_lk6_out <= #168
#170 WORD_TO_BOOL(vl_self_lk6_in)
#171 vl_self_lk6_out <= #170
#172 WORD_TO_BOOL(tros_self_lk9_in)
#173 tros_self_lk9_out <= #172
#174 WORD_TO_BOOL(shod_self_lk9_in)
#175 shod_self_lk9_out <= #174
#176 WORD_TO_BOOL(ogr_self_lk9_in)
#177 ogr_self_lk9_out <= #176
#178 WORD_TO_BOOL(vl_self_lk9_in)
#179 vl_self_lk9_out <= #178
#180 WORD_TO_BOOL(vl_self_lp1_3_in)
#181 vl_self_lp1_3_out <= #180
#182 WORD_TO_BOOL(tros_self_lk5_in)
#183 tros_self_lk5_out <= #182
#184 WORD_TO_BOOL(shod_self_lk5_in)
#185 shod_self_lk5_out <= #184
#186 WORD_TO_BOOL(ogr_self_lk5_in)
#187 ogr_self_lk5_out <= #186
#188 WORD_TO_BOOL(vl_self_lk5_in)
#189 vl_self_lk5_out <= #188
#190 WORD_TO_BOOL(revers_in)
#191 revers_out <= #190
#192 WORD_TO_BOOL(vl_self_lp4_in)
#193 vl_self_lp4_out <= #192
#194 WORD_TO_BOOL(vl_self_lp5_in)
#195 vl_self_lp5_out <= #194
#196 WORD_TO_BOOL(pusk_shnek_razg_in)
#197 pusk_shnek_razg_out <= #196
#198 WORD_TO_BOOL(stop_shnek_razg_in)
#199 stop_shnek_razg_out <= #198
#200 WORD_TO_BOOL(pusk_cyc_cleen_in)
#201 pusk_cyc_cleen_out <= #200
#202 WORD_TO_BOOL(stop_cyc_cleen_in)
#203 stop_cyc_cleen_out <= #202
_END_CFC_
(* the same logic as Structured Text *)
pusk_LAN_LP4_out := WORD_TO_BOOL(pusk_LAN_LP4);
tros_self_lk4_out := WORD_TO_BOOL(tros_self_lk4_in);
stop_LAN_LP4_out := WORD_TO_BOOL(stop_LAN_LP4);
shod_self_lk4_out := WORD_TO_BOOL(shod_self_lk4_in);
pusk_LAN_LP5_out := WORD_TO_BOOL(pusk_LAN_LP5);
vl_self_lk4_out := WORD_TO_BOOL(vl_self_lk4_in);
stop_LAN_LP5_out := WORD_TO_BOOL(stop_LAN_LP5);
tros_self_lk3_out := WORD_TO_BOOL(tros_self_lk3_in);
pusk_LAN_VP1_out := WORD_TO_BOOL(pusk_LAN_VP1);
shod_self_lk3_out := WORD_TO_BOOL(shod_self_lk3_in);
stop_LAN_VP1_out := WORD_TO_BOOL(stop_LAN_VP1);
ogr_self_lk3_out := WORD_TO_BOOL(ogr_self_lk3_in);
pusk_lan_LK10_out := WORD_TO_BOOL(pusk_lan_LK10);
vl_self_lk3_out := WORD_TO_BOOL(vl_self_lk3_in);
pusk_lan_LK11_out := WORD_TO_BOOL(pusk_lan_LK11);
tros_self_lk2_out := WORD_TO_BOOL(tros_self_lk2_in);
pusk_lan_LK12_out := WORD_TO_BOOL(pusk_lan_LK12);
shod_self_lk2_out := WORD_TO_BOOL(shod_self_lk2_in);
pusk_lan_LK13_out := WORD_TO_BOOL(pusk_lan_LK13);
ogr_self_lk2_out := WORD_TO_BOOL(ogr_self_lk2_in);
pusk_lan_GR3_out := WORD_TO_BOOL(pusk_lan_GR3);
vl_self_lk2_out := WORD_TO_BOOL(vl_self_lk2_in);
pusk_lan_LK7out := WORD_TO_BOOL(pusk_lan_LK7);
pusk_lan_LK8_out := WORD_TO_BOOL(pusk_lan_LK8);
pusk_lan_LK6_out := WORD_TO_BOOL(pusk_lan_LK6);
pusk_lan_LP1_3_out := WORD_TO_BOOL(pusk_lan_LP1_3);
pusk_lan_GR2_out := WORD_TO_BOOL(pusk_lan_GR2);
pusk_lan_LK5_out := WORD_TO_BOOL(pusk_lan_LK5);
pusk_lan_LK4_out := WORD_TO_BOOL(pusk_lan_LK4);
pusk_lan_GR1_out := WORD_TO_BOOL(pusk_lan_GR1);
pusk_lan_LK2_out := WORD_TO_BOOL(pusk_lan_LK2);
stop_lan_LK10_out := WORD_TO_BOOL(stop_lan_LK10);
stop_lan_LK11_out := WORD_TO_BOOL(stop_lan_LK11);
stop_lan_LK12_out := WORD_TO_BOOL(stop_lan_LK12);
stop_lan_LK13_out := WORD_TO_BOOL(stop_lan_LK13);
stop_lan_GR3_out := WORD_TO_BOOL(stop_lan_GR3);
stop_lan_LK7_out := WORD_TO_BOOL(stop_lan_LK7);
stop_lan_LK8_out := WORD_TO_BOOL(stop_lan_LK8);
stop_lan_LK6_out := WORD_TO_BOOL(stop_lan_LK6);
stop_lan_LK9_out := WORD_TO_BOOL(stop_lan_LK9);
stop_lan_LP1_3_out := WORD_TO_BOOL(stop_lan_LP1_3);
stop_lan_GR2_out := WORD_TO_BOOL(stop_lan_GR2);
stop_lan_LK5_out := WORD_TO_BOOL(stop_lan_LK5);
stop_lan_LK4_out := WORD_TO_BOOL(stop_lan_LK4);
stop_lan_LK3_out := WORD_TO_BOOL(stop_lan_LK3);
stop_lan_GR1_out := WORD_TO_BOOL(stop_lan_GR1);
stop_lan_LK2_out := WORD_TO_BOOL(stop_lan_LK2);
stop_LAN_D3_out := WORD_TO_BOOL(stop_LAN_D3);
stop_LAN_D4_out := WORD_TO_BOOL(stop_LAN_D4);
pusk_lan_LK9_out := WORD_TO_BOOL(pusk_lan_LK9);
pusk_lan_LK4_out := WORD_TO_BOOL(pusk_lan_LK4);
pusk_lan_D2_out := WORD_TO_BOOL(pusk_lan_D2);
stop_lan_D2_out := WORD_TO_BOOL(stop_lan_D2);
pusk_lan_D3_out := WORD_TO_BOOL(pusk_lan_D3);
pusk_lan_D4_out := WORD_TO_BOOL(pusk_lan_D4);
pusk_lan_LK3_out := WORD_TO_BOOL(pusk_lan_LK3);
pusk_lan_cyclone_out := WORD_TO_BOOL(pusk_lan_cyclone);
stop_lan_cyclone_out := WORD_TO_BOOL(stop_lan_cyclone);
tros_self_lk10_out := WORD_TO_BOOL(tros_self_lk10_in);
shod_self_lk10_out := WORD_TO_BOOL(shod_self_lk10_in);
ogr_self_lk10_out := WORD_TO_BOOL(ogr_self_lk10_in);
vl_self_lk10_out := WORD_TO_BOOL(vl_self_lk10_in);
tros_self_lk11_out := WORD_TO_BOOL(tros_self_lk11_in);
shod_self_lk11_out := WORD_TO_BOOL(shod_self_lk11_in);
ogr_self_lk11_out := WORD_TO_BOOL(ogr_self_lk11_in);
vl_self_lk11_out := WORD_TO_BOOL(vl_self_lk11_in);
tros_self_lk12_out := WORD_TO_BOOL(tros_self_lk12_in);
shod_self_lk12_out := WORD_TO_BOOL(shod_self_lk12_in);
ogr_self_lk12_out := WORD_TO_BOOL(ogr_self_lk12_in);
vl_self_lk12_out := WORD_TO_BOOL(vl_self_lk12_in);
tros_self_lk13_out := WORD_TO_BOOL(tros_self_lk13_in);
shod_self_lk13_out := WORD_TO_BOOL(shod_self_lk13_in);
ogr_self_lk13_out := WORD_TO_BOOL(ogr_self_lk13_in);
vl_self_lk13_out := WORD_TO_BOOL(vl_self_lk13_in);
tros_self_lk7_out := WORD_TO_BOOL(tros_self_lk7_in);
shod_self_lk7_out := WORD_TO_BOOL(shod_self_lk7_in);
ogr_self_lk7_out := WORD_TO_BOOL(ogr_self_lk7_in);
vl_self_lk7_out := WORD_TO_BOOL(vl_self_lk7_in);
tros_self_lk8_out := WORD_TO_BOOL(tros_self_lk8_in);
shod_self_lk8_out := WORD_TO_BOOL(shod_self_lk8_in);
ogr_self_lk8_out := WORD_TO_BOOL(ogr_self_lk8_in);
vl_self_lk8_out := WORD_TO_BOOL(vl_self_lk8_in);
tros_self_lk6_out := WORD_TO_BOOL(tros_self_lk6_in);
shod_self_lk6_out := WORD_TO_BOOL(shod_self_lk6_in);
ogr_self_lk6_out := WORD_TO_BOOL(ogr_self_lk6_in);
vl_self_lk6_out := WORD_TO_BOOL(vl_self_lk6_in);
tros_self_lk9_out := WORD_TO_BOOL(tros_self_lk9_in);
shod_self_lk9_out := WORD_TO_BOOL(shod_self_lk9_in);
ogr_self_lk9_out := WORD_TO_BOOL(ogr_self_lk9_in);
vl_self_lk9_out := WORD_TO_BOOL(vl_self_lk9_in);
vl_self_lp1_3_out := WORD_TO_BOOL(vl_self_lp1_3_in);
tros_self_lk5_out := WORD_TO_BOOL(tros_self_lk5_in);
shod_self_lk5_out := WORD_TO_BOOL(shod_self_lk5_in);
ogr_self_lk5_out := WORD_TO_BOOL(ogr_self_lk5_in);
vl_self_lk5_out := WORD_TO_BOOL(vl_self_lk5_in);
revers_out := WORD_TO_BOOL(revers_in);
vl_self_lp4_out := WORD_TO_BOOL(vl_self_lp4_in);
vl_self_lp5_out := WORD_TO_BOOL(vl_self_lp5_in);
pusk_shnek_razg_out := WORD_TO_BOOL(pusk_shnek_razg_in);
stop_shnek_razg_out := WORD_TO_BOOL(stop_shnek_razg_in);
pusk_cyc_cleen_out := WORD_TO_BOOL(pusk_cyc_cleen_in);
stop_cyc_cleen_out := WORD_TO_BOOL(stop_cyc_cleen_in);
END_FUNCTION_BLOCK

(* POU alarm_all, LD *)
FUNCTION_BLOCK alarm_all
VAR_INPUT
	err_LK10: BOOL;
	err_LK11: BOOL;
	err_LK12: BOOL;
	err_LK13: BOOL;
	err_GR3: BOOL;
	err_LK7: BOOL;
	err_LK8: BOOL;
	err_LK6: BOOL;
	err_LK9: BOOL;
	err_LP1_3_mod1: BOOL;
	err_LP1_3_mod2: BOOL;
	err_GR2: BOOL;
	err_LK5: BOOL;
	err_LP4: BOOL;
	err_LP5: BOOL;
	err_LK4: BOOL;
	err_GR1: BOOL;
	err_LK2: BOOL;
	err_LK3: BOOL;
	err_VP1: BOOL;
	err_D3_mod1: BOOL;
	err_D3_mod2: BOOL;
	err_D4_mod1: BOOL;
	err_D4_mod2: BOOL;
	err_D2: BOOL;
	err_cyc1: BOOL;
	err_cyc2: BOOL;
	err_lp4_temp: BOOL;
	err_d3_temp: BOOL;
	err_d4_temp: BOOL;
	err_vp1_temp: BOOL;
END_VAR
VAR_OUTPUT
	modul_out: BOOL;
END_VAR
VAR
END_VAR
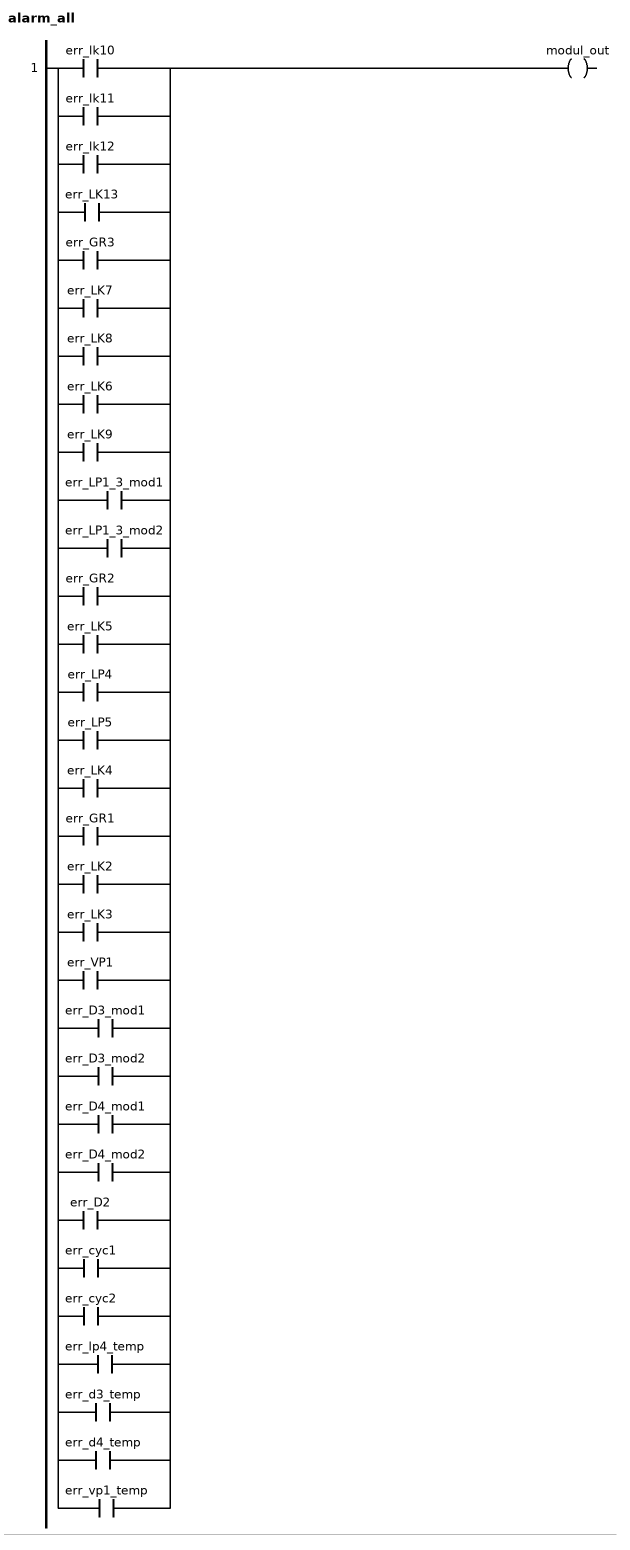
_LD_ (* Ladder Diagram *)
NETWORK 1
	{ [err_lk10] | [err_lk11] | [err_lk12] | [err_LK13] | [err_GR3] | [err_LK7] | [err_LK8] | [err_LK6] | [err_LK9] | [err_LP1_3_mod1] | [err_LP1_3_mod2] | [err_GR2] | [err_LK5] | [err_LP4] | [err_LP5] | [err_LK4] | [err_GR1] | [err_LK2] | [err_LK3] | [err_VP1] | [err_D3_mod1] | [err_D3_mod2] | [err_D4_mod1] | [err_D4_mod2] | [err_D2] | [err_cyc1] | [err_cyc2] | [err_lp4_temp] | [err_d3_temp] | [err_d4_temp] | [err_vp1_temp] } --- (modul_out)
_END_LD_
(* the same logic as Structured Text *)
(* Network 1 *)
modul_out := err_lk10 OR err_lk11 OR err_lk12 OR err_LK13 OR err_GR3 OR err_LK7 OR err_LK8 OR err_LK6 OR err_LK9 OR err_LP1_3_mod1 OR err_LP1_3_mod2 OR err_GR2 OR err_LK5 OR err_LP4 OR err_LP5 OR err_LK4 OR err_GR1 OR err_LK2 OR err_LK3 OR err_VP1 OR err_D3_mod1 OR err_D3_mod2 OR err_D4_mod1 OR err_D4_mod2 OR err_D2 OR err_cyc1 OR err_cyc2 OR err_lp4_temp OR err_d3_temp OR err_d4_temp OR err_vp1_temp;
END_FUNCTION_BLOCK

(* POU if_LV, ST *)
FUNCTION_BLOCK if_LV
VAR_INPUT
	input_LV2_LK7: REAL;
	input_LV1_LK7: REAL;
	input_LV2_LK8: REAL;
	input_LV1_LK8: REAL;
	input_LV2_GR1: REAL;
	input_LV1_GR1: REAL;
	input_LV2_D2: REAL;
	input_LV1_D2: REAL;
	input_time_VL: WORD;
END_VAR
VAR_OUTPUT
	output_LV2_LK7: REAL;
	output_LV1_LK7: REAL;
	output_LV2_LK8: REAL;
	output_LV1_LK8: REAL;
	output_LV2_GR1: REAL;
	output_LV1_GR1: REAL;
	output_LV2_D2: REAL;
	output_LV1_D2: REAL;
	output_time_VL: WORD;
END_VAR
VAR
END_VAR
IF input_LV2_LK7 <= 0
THEN output_LV2_LK7 := 3;
ELSE output_LV2_LK7 := input_LV2_LK7;
END_IF;

IF input_LV1_LK7 <= 0
THEN output_LV1_LK7 := 2.5;
ELSE output_LV1_LK7 := input_LV1_LK7;
END_IF;

IF input_LV2_LK8 <= 0
THEN output_LV2_LK8 := 3;
ELSE output_LV2_LK8 := input_LV2_LK8;
END_IF;

IF input_LV1_LK8 <= 0
THEN output_LV1_LK8 := 2.5;
ELSE output_LV1_LK8 := input_LV1_LK8;
END_IF;

IF input_LV2_GR1 <= 0
THEN output_LV2_GR1 := 3;
ELSE output_LV2_GR1 := input_LV2_GR1;
END_IF;

IF input_LV1_GR1 <= 0
THEN output_LV1_GR1 := 2.5;
ELSE output_LV1_GR1 := input_LV1_GR1;
END_IF;

IF input_LV2_D2 <= 0
THEN output_LV2_D2 := 2;
ELSE output_LV2_D2 := input_LV2_D2;
END_IF;

IF input_LV1_D2 <= 0
THEN output_LV1_D2 := 1.9;
ELSE output_LV1_D2 := input_LV1_D2;
END_IF;

IF input_time_VL <= 0
THEN output_time_VL := 3;
ELSE output_time_VL := input_time_VL;
END_IF;
END_FUNCTION_BLOCK

(* POU washer, LD *)
FUNCTION_BLOCK washer
VAR_INPUT
END_VAR
VAR_OUTPUT
END_VAR
VAR
END_VAR
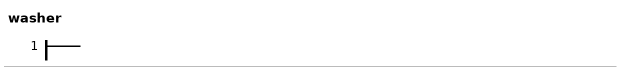
_LD_ (* Ladder Diagram *)
NETWORK 1
	*
_END_LD_
(* the same logic as Structured Text *)
(* Network 1 *)
END_FUNCTION_BLOCK
